            ! Raise pen
            MoveL Offs(next_target, x_offset, y_offset, penup_offset),approach_speed,fine,Alex_Pen_ABB\WObj:=WorkSurface;
        ELSEIF character = "j" THEN
            ! Raise pen to avoid drawing of surface
            position := Lower_J_PtA{1} * font_size;
            next_target.trans := position;
            MoveJ Offs(next_target, x_offset, y_offset, penup_offset),approach_speed,fine,Alex_Pen_ABB\WObj:=WorkSurface;

            ! Drop pen
            MoveL Offs(next_target, x_offset, y_offset, z_offset),approach_speed,fine,Alex_Pen_ABB\WObj:=WorkSurface;

            FOR index FROM 1 TO Dim(Lower_J_PtA, 1) DO
                position := Lower_J_PtA{index} * font_size;
                next_target.trans := position; last_index := index;

                MoveJ Offs(next_target, x_offset, y_offset, z_offset),write_speed,fine,Alex_Pen_ABB\WObj:=WorkSurface;
            ENDFOR

            ! Raise pen
            MoveL Offs(next_target, x_offset, y_offset, penup_offset),approach_speed,fine,Alex_Pen_ABB\WObj:=WorkSurface;

            ! Raise pen to avoid drawing of surface
            position := Lower_J_PtB{1} * font_size;
            next_target.trans := position;
            MoveJ Offs(next_target, x_offset, y_offset, penup_offset),approach_speed,fine,Alex_Pen_ABB\WObj:=WorkSurface;

            ! Drop pen
            MoveL Offs(next_target, x_offset, y_offset, z_offset),approach_speed,fine,Alex_Pen_ABB\WObj:=WorkSurface;

            FOR index FROM 1 TO Dim(Lower_J_PtB, 1) DO
                position := Lower_J_PtB{index} * font_size;
                next_target.trans := position; last_index := index;

                MoveJ Offs(next_target, x_offset, y_offset, z_offset),write_speed,fine,Alex_Pen_ABB\WObj:=WorkSurface;
            ENDFOR

            ! Raise pen
            MoveL Offs(next_target, x_offset, y_offset, penup_offset),approach_speed,fine,Alex_Pen_ABB\WObj:=WorkSurface;
        ELSEIF character = "k" THEN
            ! Raise pen to avoid drawing of surface
            position := Lower_K_PtA{1} * font_size;
            next_target.trans := position;
            MoveJ Offs(next_target, x_offset, y_offset, penup_offset),approach_speed,fine,Alex_Pen_ABB\WObj:=WorkSurface;

            ! Drop pen
            MoveL Offs(next_target, x_offset, y_offset, z_offset),approach_speed,fine,Alex_Pen_ABB\WObj:=WorkSurface;

            FOR index FROM 1 TO Dim(Lower_K_PtA, 1) DO
                position := Lower_K_PtA{index} * font_size;
                next_target.trans := position; last_index := index;

                MoveJ Offs(next_target, x_offset, y_offset, z_offset),write_speed,fine,Alex_Pen_ABB\WObj:=WorkSurface;
            ENDFOR

            ! Raise pen
            MoveL Offs(next_target, x_offset, y_offset, penup_offset),approach_speed,fine,Alex_Pen_ABB\WObj:=WorkSurface;
        ELSEIF character = "l" THEN
            ! Raise pen to avoid drawing of surface
            position := Lower_L_PtA{1} * font_size;
            next_target.trans := position;
            MoveJ Offs(next_target, x_offset, y_offset, penup_offset),approach_speed,fine,Alex_Pen_ABB\WObj:=WorkSurface;

            ! Drop pen
            MoveL Offs(next_target, x_offset, y_offset, z_offset),approach_speed,fine,Alex_Pen_ABB\WObj:=WorkSurface;

            FOR index FROM 1 TO Dim(Lower_L_PtA, 1) DO
                position := Lower_L_PtA{index} * font_size;
                next_target.trans := position; last_index := index;

                MoveJ Offs(next_target, x_offset, y_offset, z_offset),write_speed,fine,Alex_Pen_ABB\WObj:=WorkSurface;
            ENDFOR

            ! Raise pen
            MoveL Offs(next_target, x_offset, y_offset, penup_offset),approach_speed,fine,Alex_Pen_ABB\WObj:=WorkSurface;
        ELSEIF character = "m" THEN
            ! Raise pen to avoid drawing of surface
            position := Lower_M_PtA{1} * font_size;
            next_target.trans := position;
            MoveJ Offs(next_target, x_offset, y_offset, penup_offset),approach_speed,fine,Alex_Pen_ABB\WObj:=WorkSurface;

            ! Drop pen
            MoveL Offs(next_target, x_offset, y_offset, z_offset),approach_speed,fine,Alex_Pen_ABB\WObj:=WorkSurface;

            FOR index FROM 1 TO Dim(Lower_M_PtA, 1) DO
                position := Lower_M_PtA{index} * font_size;
                next_target.trans := position; last_index := index;

                MoveJ Offs(next_target, x_offset, y_offset, z_offset),write_speed,fine,Alex_Pen_ABB\WObj:=WorkSurface;
            ENDFOR

            ! Raise pen
            MoveL Offs(next_target, x_offset, y_offset, penup_offset),approach_speed,fine,Alex_Pen_ABB\WObj:=WorkSurface;
        ELSEIF character = "n" THEN
            ! Raise pen to avoid drawing of surface
            position := Lower_N_PtA{1} * font_size;
            next_target.trans := position;
            MoveJ Offs(next_target, x_offset, y_offset, penup_offset),approach_speed,fine,Alex_Pen_ABB\WObj:=WorkSurface;

            ! Drop pen
            MoveL Offs(next_target, x_offset, y_offset, z_offset),approach_speed,fine,Alex_Pen_ABB\WObj:=WorkSurface;

            FOR index FROM 1 TO Dim(Lower_N_PtA, 1) DO
                position := Lower_N_PtA{index} * font_size;
                next_target.trans := position; last_index := index;

                MoveJ Offs(next_target, x_offset, y_offset, z_offset),write_speed,fine,Alex_Pen_ABB\WObj:=WorkSurface;
            ENDFOR

            ! Raise pen
            MoveL Offs(next_target, x_offset, y_offset, penup_offset),approach_speed,fine,Alex_Pen_ABB\WObj:=WorkSurface;
        ELSEIF character = "o" THEN
            ! Raise pen to avoid drawing of surface
            position := Lower_O_PtA{1} * font_size;
            next_target.trans := position;
            MoveJ Offs(next_target, x_offset, y_offset, penup_offset),approach_speed,fine,Alex_Pen_ABB\WObj:=WorkSurface;

            ! Drop pen
            MoveL Offs(next_target, x_offset, y_offset, z_offset),approach_speed,fine,Alex_Pen_ABB\WObj:=WorkSurface;

            FOR index FROM 1 TO Dim(Lower_O_PtA, 1) DO
                position := Lower_O_PtA{index} * font_size;
                next_target.trans := position; last_index := index;

                MoveJ Offs(next_target, x_offset, y_offset, z_offset),write_speed,fine,Alex_Pen_ABB\WObj:=WorkSurface;
            ENDFOR

            ! Raise pen
            MoveL Offs(next_target, x_offset, y_offset, penup_offset),approach_speed,fine,Alex_Pen_ABB\WObj:=WorkSurface;

            ! Raise pen to avoid drawing of surface
            position := Lower_O_PtB{1} * font_size;
            next_target.trans := position;
            MoveJ Offs(next_target, x_offset, y_offset, penup_offset),approach_speed,fine,Alex_Pen_ABB\WObj:=WorkSurface;

            ! Drop pen
            MoveL Offs(next_target, x_offset, y_offset, z_offset),approach_speed,fine,Alex_Pen_ABB\WObj:=WorkSurface;

            FOR index FROM 1 TO Dim(Lower_O_PtB, 1) DO
                position := Lower_O_PtB{index} * font_size;
                next_target.trans := position; last_index := index;

                MoveJ Offs(next_target, x_offset, y_offset, z_offset),write_speed,fine,Alex_Pen_ABB\WObj:=WorkSurface;
            ENDFOR

            ! Raise pen
            MoveL Offs(next_target, x_offset, y_offset, penup_offset),approach_speed,fine,Alex_Pen_ABB\WObj:=WorkSurface;
        ELSEIF character = "p" THEN
            ! Raise pen to avoid drawing of surface
            position := Lower_P_PtA{1} * font_size;
            next_target.trans := position;
            MoveJ Offs(next_target, x_offset, y_offset, penup_offset),approach_speed,fine,Alex_Pen_ABB\WObj:=WorkSurface;

            ! Drop pen
            MoveL Offs(next_target, x_offset, y_offset, z_offset),approach_speed,fine,Alex_Pen_ABB\WObj:=WorkSurface;

            FOR index FROM 1 TO Dim(Lower_P_PtA, 1) DO
                position := Lower_P_PtA{index} * font_size;
                next_target.trans := position; last_index := index;

                MoveJ Offs(next_target, x_offset, y_offset, z_offset),write_speed,fine,Alex_Pen_ABB\WObj:=WorkSurface;
            ENDFOR

            ! Raise pen
            MoveL Offs(next_target, x_offset, y_offset, penup_offset),approach_speed,fine,Alex_Pen_ABB\WObj:=WorkSurface;

            ! Raise pen to avoid drawing of surface
            position := Lower_P_PtB{1} * font_size;
            next_target.trans := position;
            MoveJ Offs(next_target, x_offset, y_offset, penup_offset),approach_speed,fine,Alex_Pen_ABB\WObj:=WorkSurface;

            ! Drop pen
            MoveL Offs(next_target, x_offset, y_offset, z_offset),approach_speed,fine,Alex_Pen_ABB\WObj:=WorkSurface;

            FOR index FROM 1 TO Dim(Lower_P_PtB, 1) DO
                position := Lower_P_PtB{index} * font_size;
                next_target.trans := position; last_index := index;

                MoveJ Offs(next_target, x_offset, y_offset, z_offset),write_speed,fine,Alex_Pen_ABB\WObj:=WorkSurface;
            ENDFOR

            ! Raise pen
            MoveL Offs(next_target, x_offset, y_offset, penup_offset),approach_speed,fine,Alex_Pen_ABB\WObj:=WorkSurface;
        ELSEIF character = "q" THEN
            ! Raise pen to avoid drawing of surface
            position := Lower_Q_PtA{1} * font_size;
            next_target.trans := position;
            MoveJ Offs(next_target, x_offset, y_offset, penup_offset),approach_speed,fine,Alex_Pen_ABB\WObj:=WorkSurface;

            ! Drop pen
            MoveL Offs(next_target, x_offset, y_offset, z_offset),approach_speed,fine,Alex_Pen_ABB\WObj:=WorkSurface;

            FOR index FROM 1 TO Dim(Lower_Q_PtA, 1) DO
                position := Lower_Q_PtA{index} * font_size;
                next_target.trans := position; last_index := index;

                MoveJ Offs(next_target, x_offset, y_offset, z_offset),write_speed,fine,Alex_Pen_ABB\WObj:=WorkSurface;
            ENDFOR

            ! Raise pen
            MoveL Offs(next_target, x_offset, y_offset, penup_offset),approach_speed,fine,Alex_Pen_ABB\WObj:=WorkSurface;

            ! Raise pen to avoid drawing of surface
            position := Lower_Q_PtB{1} * font_size;
            next_target.trans := position;
            MoveJ Offs(next_target, x_offset, y_offset, penup_offset),approach_speed,fine,Alex_Pen_ABB\WObj:=WorkSurface;

            ! Drop pen
            MoveL Offs(next_target, x_offset, y_offset, z_offset),approach_speed,fine,Alex_Pen_ABB\WObj:=WorkSurface;

            FOR index FROM 1 TO Dim(Lower_Q_PtB, 1) DO
                position := Lower_Q_PtB{index} * font_size;
                next_target.trans := position; last_index := index;

                MoveJ Offs(next_target, x_offset, y_offset, z_offset),write_speed,fine,Alex_Pen_ABB\WObj:=WorkSurface;
            ENDFOR

            ! Raise pen
            MoveL Offs(next_target, x_offset, y_offset, penup_offset),approach_speed,fine,Alex_Pen_ABB\WObj:=WorkSurface;
        ELSEIF character = "r" THEN
            ! Raise pen to avoid drawing of surface
            position := Lower_R_PtA{1} * font_size;
            next_target.trans := position;
            MoveJ Offs(next_target, x_offset, y_offset, penup_offset),approach_speed,fine,Alex_Pen_ABB\WObj:=WorkSurface;

            ! Drop pen
            MoveL Offs(next_target, x_offset, y_offset, z_offset),approach_speed,fine,Alex_Pen_ABB\WObj:=WorkSurface;

            FOR index FROM 1 TO Dim(Lower_R_PtA, 1) DO
                position := Lower_R_PtA{index} * font_size;
                next_target.trans := position; last_index := index;

                MoveJ Offs(next_target, x_offset, y_offset, z_offset),write_speed,fine,Alex_Pen_ABB\WObj:=WorkSurface;
            ENDFOR

            ! Raise pen
            MoveL Offs(next_target, x_offset, y_offset, penup_offset),approach_speed,fine,Alex_Pen_ABB\WObj:=WorkSurface;
        ELSEIF character = "s" THEN
            ! Raise pen to avoid drawing of surface
            position := Lower_S_PtA{1} * font_size;
            next_target.trans := position;
            MoveJ Offs(next_target, x_offset, y_offset, penup_offset),approach_speed,fine,Alex_Pen_ABB\WObj:=WorkSurface;

            ! Drop pen
            MoveL Offs(next_target, x_offset, y_offset, z_offset),approach_speed,fine,Alex_Pen_ABB\WObj:=WorkSurface;

            FOR index FROM 1 TO Dim(Lower_S_PtA, 1) DO
                position := Lower_S_PtA{index} * font_size;
                next_target.trans := position; last_index := index;

                MoveJ Offs(next_target, x_offset, y_offset, z_offset),write_speed,fine,Alex_Pen_ABB\WObj:=WorkSurface;
            ENDFOR

            ! Raise pen
            MoveL Offs(next_target, x_offset, y_offset, penup_offset),approach_speed,fine,Alex_Pen_ABB\WObj:=WorkSurface;
        ELSEIF character = "t" THEN
            ! Raise pen to avoid drawing of surface
            position := Lower_T_PtA{1} * font_size;
            next_target.trans := position;
            MoveJ Offs(next_target, x_offset, y_offset, penup_offset),approach_speed,fine,Alex_Pen_ABB\WObj:=WorkSurface;

            ! Drop pen
            MoveL Offs(next_target, x_offset, y_offset, z_offset),approach_speed,fine,Alex_Pen_ABB\WObj:=WorkSurface;

            FOR index FROM 1 TO Dim(Lower_T_PtA, 1) DO
                position := Lower_T_PtA{index} * font_size;
                next_target.trans := position; last_index := index;

                MoveJ Offs(next_target, x_offset, y_offset, z_offset),write_speed,fine,Alex_Pen_ABB\WObj:=WorkSurface;
            ENDFOR

            ! Raise pen
            MoveL Offs(next_target, x_offset, y_offset, penup_offset),approach_speed,fine,Alex_Pen_ABB\WObj:=WorkSurface;
        ELSEIF character = "u" THEN
            ! Raise pen to avoid drawing of surface
            position := Lower_U_PtA{1} * font_size;
            next_target.trans := position;
            MoveJ Offs(next_target, x_offset, y_offset, penup_offset),approach_speed,fine,Alex_Pen_ABB\WObj:=WorkSurface;

            ! Drop pen
            MoveL Offs(next_target, x_offset, y_offset, z_offset),approach_speed,fine,Alex_Pen_ABB\WObj:=WorkSurface;

            FOR index FROM 1 TO Dim(Lower_U_PtA, 1) DO
                position := Lower_U_PtA{index} * font_size;
                next_target.trans := position; last_index := index;

                MoveJ Offs(next_target, x_offset, y_offset, z_offset),write_speed,fine,Alex_Pen_ABB\WObj:=WorkSurface;
            ENDFOR

            ! Raise pen
            MoveL Offs(next_target, x_offset, y_offset, penup_offset),approach_speed,fine,Alex_Pen_ABB\WObj:=WorkSurface;
        ELSEIF character = "v" THEN
            ! Raise pen to avoid drawing of surface
            position := Lower_V_PtA{1} * font_size;
            next_target.trans := position;
            MoveJ Offs(next_target, x_offset, y_offset, penup_offset),approach_speed,fine,Alex_Pen_ABB\WObj:=WorkSurface;

            ! Drop pen
            MoveL Offs(next_target, x_offset, y_offset, z_offset),approach_speed,fine,Alex_Pen_ABB\WObj:=WorkSurface;

            FOR index FROM 1 TO Dim(Lower_V_PtA, 1) DO
                position := Lower_V_PtA{index} * font_size;
                next_target.trans := position; last_index := index;

                MoveJ Offs(next_target, x_offset, y_offset, z_offset),write_speed,fine,Alex_Pen_ABB\WObj:=WorkSurface;
            ENDFOR

            ! Raise pen
            MoveL Offs(next_target, x_offset, y_offset, penup_offset),approach_speed,fine,Alex_Pen_ABB\WObj:=WorkSurface;
        ELSEIF character = "w" THEN
            ! Raise pen to avoid drawing of surface
            position := Lower_W_PtA{1} * font_size;
            next_target.trans := position;
            MoveJ Offs(next_target, x_offset, y_offset, penup_offset),approach_speed,fine,Alex_Pen_ABB\WObj:=WorkSurface;

            ! Drop pen
            MoveL Offs(next_target, x_offset, y_offset, z_offset),approach_speed,fine,Alex_Pen_ABB\WObj:=WorkSurface;

            FOR index FROM 1 TO Dim(Lower_W_PtA, 1) DO
                position := Lower_W_PtA{index} * font_size;
                next_target.trans := position; last_index := index;

                MoveJ Offs(next_target, x_offset, y_offset, z_offset),write_speed,fine,Alex_Pen_ABB\WObj:=WorkSurface;
            ENDFOR

            ! Raise pen
            MoveL Offs(next_target, x_offset, y_offset, penup_offset),approach_speed,fine,Alex_Pen_ABB\WObj:=WorkSurface;
        ELSEIF character = "x" THEN
            ! Raise pen to avoid drawing of surface
            position := Lower_X_PtA{1} * font_size;
            next_target.trans := position;
            MoveJ Offs(next_target, x_offset, y_offset, penup_offset),approach_speed,fine,Alex_Pen_ABB\WObj:=WorkSurface;

            ! Drop pen
            MoveL Offs(next_target, x_offset, y_offset, z_offset),approach_speed,fine,Alex_Pen_ABB\WObj:=WorkSurface;

            FOR index FROM 1 TO Dim(Lower_X_PtA, 1) DO
                position := Lower_X_PtA{index} * font_size;
                next_target.trans := position; last_index := index;

                MoveJ Offs(next_target, x_offset, y_offset, z_offset),write_speed,fine,Alex_Pen_ABB\WObj:=WorkSurface;
            ENDFOR

            ! Raise pen
            MoveL Offs(next_target, x_offset, y_offset, penup_offset),approach_speed,fine,Alex_Pen_ABB\WObj:=WorkSurface;
        ELSEIF character = "y" THEN
            ! Raise pen to avoid drawing of surface
            position := Lower_Y_PtA{1} * font_size;
            next_target.trans := position;
            MoveJ Offs(next_target, x_offset, y_offset, penup_offset),approach_speed,fine,Alex_Pen_ABB\WObj:=WorkSurface;

            ! Drop pen
            MoveL Offs(next_target, x_offset, y_offset, z_offset),approach_speed,fine,Alex_Pen_ABB\WObj:=WorkSurface;

            FOR index FROM 1 TO Dim(Lower_Y_PtA, 1) DO
                position := Lower_Y_PtA{index} * font_size;
                next_target.trans := position; last_index := index;

                MoveJ Offs(next_target, x_offset, y_offset, z_offset),write_speed,fine,Alex_Pen_ABB\WObj:=WorkSurface;
            ENDFOR

            ! Raise pen
            MoveL Offs(next_target, x_offset, y_offset, penup_offset),approach_speed,fine,Alex_Pen_ABB\WObj:=WorkSurface;
        ELSEIF character = "z" THEN
            ! Raise pen to avoid drawing of surface
            position := Lower_Z_PtA{1} * font_size;
            next_target.trans := position;
            MoveJ Offs(next_target, x_offset, y_offset, penup_offset),approach_speed,fine,Alex_Pen_ABB\WObj:=WorkSurface;

            ! Drop pen
            MoveL Offs(next_target, x_offset, y_offset, z_offset),approach_speed,fine,Alex_Pen_ABB\WObj:=WorkSurface;

            FOR index FROM 1 TO Dim(Lower_Z_PtA, 1) DO
                position := Lower_Z_PtA{index} * font_size;
                next_target.trans := position; last_index := index;

                MoveJ Offs(next_target, x_offset, y_offset, z_offset),write_speed,fine,Alex_Pen_ABB\WObj:=WorkSurface;
            ENDFOR

            ! Raise pen
            MoveL Offs(next_target, x_offset, y_offset, penup_offset),approach_speed,fine,Alex_Pen_ABB\WObj:=WorkSurface;
        ELSEIF character = "{" THEN
            ! Raise pen to avoid drawing of surface
            position := OpenCurlyBrackets_PtA{1} * font_size;
            next_target.trans := position;
            MoveJ Offs(next_target, x_offset, y_offset, penup_offset),approach_speed,fine,Alex_Pen_ABB\WObj:=WorkSurface;

            ! Drop pen
            MoveL Offs(next_target, x_offset, y_offset, z_offset),approach_speed,fine,Alex_Pen_ABB\WObj:=WorkSurface;

            FOR index FROM 1 TO Dim(OpenCurlyBrackets_PtA, 1) DO
                position := OpenCurlyBrackets_PtA{index} * font_size;
                next_target.trans := position; last_index := index;

                MoveJ Offs(next_target, x_offset, y_offset, z_offset),write_speed,fine,Alex_Pen_ABB\WObj:=WorkSurface;
            ENDFOR

            ! Raise pen
            MoveL Offs(next_target, x_offset, y_offset, penup_offset),approach_speed,fine,Alex_Pen_ABB\WObj:=WorkSurface;
        ELSEIF character = "}" THEN
            ! Raise pen to avoid drawing of surface
            position := CloseCurlyBrackets_PtB{1} * font_size;
            next_target.trans := position;
            MoveJ Offs(next_target, x_offset, y_offset, penup_offset),approach_speed,fine,Alex_Pen_ABB\WObj:=WorkSurface;

            ! Drop pen
            MoveL Offs(next_target, x_offset, y_offset, z_offset),approach_speed,fine,Alex_Pen_ABB\WObj:=WorkSurface;

            FOR index FROM 1 TO Dim(CloseCurlyBrackets_PtB, 1) DO
                position := CloseCurlyBrackets_PtB{index} * font_size;
                next_target.trans := position; last_index := index;

                MoveJ Offs(next_target, x_offset, y_offset, z_offset),write_speed,fine,Alex_Pen_ABB\WObj:=WorkSurface;
            ENDFOR

            ! Raise pen
            MoveL Offs(next_target, x_offset, y_offset, penup_offset),approach_speed,fine,Alex_Pen_ABB\WObj:=WorkSurface;
        ELSEIF character = "|" THEN
            ! Raise pen to avoid drawing of surface
            position := VerticalBar_PtA{1} * font_size;
            next_target.trans := position;
            MoveJ Offs(next_target, x_offset, y_offset, penup_offset),approach_speed,fine,Alex_Pen_ABB\WObj:=WorkSurface;

            ! Drop pen
            MoveL Offs(next_target, x_offset, y_offset, z_offset),approach_speed,fine,Alex_Pen_ABB\WObj:=WorkSurface;

            FOR index FROM 1 TO Dim(VerticalBar_PtA, 1) DO
                position := VerticalBar_PtA{index} * font_size;
                next_target.trans := position; last_index := index;

                MoveJ Offs(next_target, x_offset, y_offset, z_offset),write_speed,fine,Alex_Pen_ABB\WObj:=WorkSurface;
            ENDFOR

            ! Raise pen
            MoveL Offs(next_target, x_offset, y_offset, penup_offset),approach_speed,fine,Alex_Pen_ABB\WObj:=WorkSurface;
        ELSEIF character = "~" THEN
            ! Raise pen to avoid drawing of surface
            position := Tilty_PtA{1} * font_size;
            next_target.trans := position;
            MoveJ Offs(next_target, x_offset, y_offset, penup_offset),approach_speed,fine,Alex_Pen_ABB\WObj:=WorkSurface;

            ! Drop pen
            MoveL Offs(next_target, x_offset, y_offset, z_offset),approach_speed,fine,Alex_Pen_ABB\WObj:=WorkSurface;

            FOR index FROM 1 TO Dim(Tilty_PtA, 1) DO
                position := Tilty_PtA{index} * font_size;
                next_target.trans := position; last_index := index;

                MoveJ Offs(next_target, x_offset, y_offset, z_offset),write_speed,fine,Alex_Pen_ABB\WObj:=WorkSurface;
            ENDFOR

            ! Raise pen
            MoveL Offs(next_target, x_offset, y_offset, penup_offset),approach_speed,fine,Alex_Pen_ABB\WObj:=WorkSurface;
        ELSE
            TPWrite "Unknown character " + character;
        ENDIF

    ENDPROC


    !***********************************************************
    !
    ! Procedure DrawArtWork_House
    !   This procedure draws my house artwork on the work surface
    !   This is mainly used by the Special User function
    !
    ! Example
    !   VAR speeddata approach_speed := v100;  // Approach speed for arm
    !   VAR speeddata write_speed := v80;      // Write speed for arm
    !   VAR num x_offset := 0;                 // x offset from worksurface origin
    !   VAR num y_offset := 0;                 // y offset from worksurface origin
    !   VAR num z_offset := 0;                 // z offset from worksurface origin
    !   VAR num pen_offset := 30;              // Defines pen position for pen up
    !
    !   DrawArtWork_House 1.0, approach_speed, write_speed, x_offset, y_offset, z_offset, penup_offset;
    !
    !***********************************************************
    PROC DrawArtWork_House(num font_size, speeddata approach_speed, speeddata write_speed, num x_offset, num y_offset, num z_offset, num penup_offset)
        ! Define all points for artwork
        VAR pos pos0{30} := [[147.0, 28.0, 0],[146.0, 29.0, 0],[146.0, 48.0, 0],[147.0, 49.0, 0],[147.0, 60.0, 0],[148.0, 61.0, 0],[148.0, 67.0, 0],[149.0, 68.0, 0],[149.0, 77.0, 0],[151.0, 79.0, 0],[153.0, 79.0, 0],[154.0, 78.0, 0],[155.0, 78.0, 0],[156.0, 77.0, 0],[156.0, 72.0, 0],[155.0, 71.0, 0],[155.0, 67.0, 0],[154.0, 66.0, 0],[154.0, 60.0, 0],[153.0, 59.0, 0],[153.0, 16.0, 0],[154.0, 15.0, 0],[154.0, 13.0, 0],[151.0, 10.0, 0],[150.0, 10.0, 0],[148.0, 12.0, 0],[148.0, 14.0, 0],[147.0, 15.0, 0],[147.0, 28.0, 0],[146.0, 29.0, 0]];
        VAR pos pos1{120} := [[99.0, 127.0, 0],[98.0, 128.0, 0],[98.0, 129.0, 0],[101.0, 132.0, 0],[102.0, 131.0, 0],[103.0, 131.0, 0],[106.0, 128.0, 0],[107.0, 128.0, 0],[110.0, 125.0, 0],[111.0, 125.0, 0],[114.0, 122.0, 0],[115.0, 122.0, 0],[118.0, 119.0, 0],[119.0, 119.0, 0],[121.0, 117.0, 0],[122.0, 117.0, 0],[125.0, 114.0, 0],[126.0, 114.0, 0],[129.0, 111.0, 0],[130.0, 111.0, 0],[131.0, 110.0, 0],[132.0, 110.0, 0],[134.0, 108.0, 0],[135.0, 108.0, 0],[138.0, 105.0, 0],[139.0, 105.0, 0],[140.0, 104.0, 0],[141.0, 104.0, 0],[142.0, 103.0, 0],[143.0, 103.0, 0],[146.0, 100.0, 0],[147.0, 100.0, 0],[148.0, 99.0, 0],[149.0, 99.0, 0],[151.0, 97.0, 0],[152.0, 97.0, 0],[153.0, 96.0, 0],[154.0, 96.0, 0],[156.0, 94.0, 0],[158.0, 94.0, 0],[159.0, 93.0, 0],[159.0, 92.0, 0],[161.0, 92.0, 0],[164.0, 89.0, 0],[166.0, 89.0, 0],[168.0, 87.0, 0],[169.0, 87.0, 0],[170.0, 86.0, 0],[172.0, 86.0, 0],[175.0, 83.0, 0],[177.0, 83.0, 0],[179.0, 81.0, 0],[180.0, 81.0, 0],[181.0, 80.0, 0],[183.0, 80.0, 0],[184.0, 79.0, 0],[184.0, 78.0, 0],[186.0, 78.0, 0],[187.0, 77.0, 0],[187.0, 76.0, 0],[184.0, 73.0, 0],[182.0, 73.0, 0],[181.0, 74.0, 0],[179.0, 74.0, 0],[177.0, 76.0, 0],[176.0, 76.0, 0],[175.0, 77.0, 0],[173.0, 77.0, 0],[172.0, 78.0, 0],[172.0, 79.0, 0],[170.0, 79.0, 0],[169.0, 80.0, 0],[168.0, 80.0, 0],[166.0, 82.0, 0],[164.0, 82.0, 0],[162.0, 84.0, 0],[161.0, 84.0, 0],[160.0, 85.0, 0],[159.0, 85.0, 0],[156.0, 88.0, 0],[154.0, 88.0, 0],[151.0, 91.0, 0],[150.0, 91.0, 0],[149.0, 92.0, 0],[148.0, 92.0, 0],[147.0, 93.0, 0],[146.0, 93.0, 0],[143.0, 96.0, 0],[141.0, 96.0, 0],[138.0, 99.0, 0],[136.0, 99.0, 0],[135.0, 100.0, 0],[135.0, 101.0, 0],[134.0, 101.0, 0],[133.0, 102.0, 0],[132.0, 102.0, 0],[130.0, 104.0, 0],[129.0, 104.0, 0],[126.0, 107.0, 0],[125.0, 107.0, 0],[124.0, 108.0, 0],[123.0, 108.0, 0],[121.0, 110.0, 0],[120.0, 110.0, 0],[119.0, 111.0, 0],[119.0, 112.0, 0],[118.0, 112.0, 0],[117.0, 113.0, 0],[116.0, 113.0, 0],[113.0, 116.0, 0],[112.0, 116.0, 0],[110.0, 118.0, 0],[109.0, 118.0, 0],[105.0, 122.0, 0],[104.0, 122.0, 0],[102.0, 124.0, 0],[101.0, 124.0, 0],[99.0, 126.0, 0],[99.0, 127.0, 0],[98.0, 128.0, 0]];
        VAR pos pos2{51} := [[78.0, 87.0, 0],[78.0, 89.0, 0],[79.0, 90.0, 0],[80.0, 90.0, 0],[81.0, 91.0, 0],[82.0, 91.0, 0],[83.0, 92.0, 0],[83.0, 93.0, 0],[84.0, 94.0, 0],[84.0, 95.0, 0],[85.0, 96.0, 0],[85.0, 97.0, 0],[90.0, 102.0, 0],[91.0, 102.0, 0],[92.0, 103.0, 0],[93.0, 103.0, 0],[94.0, 104.0, 0],[96.0, 104.0, 0],[97.0, 105.0, 0],[103.0, 105.0, 0],[104.0, 104.0, 0],[105.0, 104.0, 0],[106.0, 103.0, 0],[109.0, 103.0, 0],[112.0, 100.0, 0],[113.0, 100.0, 0],[114.0, 99.0, 0],[114.0, 97.0, 0],[115.0, 97.0, 0],[116.0, 96.0, 0],[116.0, 95.0, 0],[117.0, 94.0, 0],[117.0, 92.0, 0],[118.0, 92.0, 0],[119.0, 91.0, 0],[121.0, 91.0, 0],[122.0, 90.0, 0],[122.0, 87.0, 0],[121.0, 86.0, 0],[118.0, 86.0, 0],[117.0, 87.0, 0],[111.0, 87.0, 0],[110.0, 88.0, 0],[95.0, 88.0, 0],[94.0, 87.0, 0],[86.0, 87.0, 0],[85.0, 86.0, 0],[81.0, 86.0, 0],[80.0, 85.0, 0],[78.0, 87.0, 0],[78.0, 89.0, 0]];
        VAR pos pos3{12} := [[88.0, 92.0, 0],[112.0, 92.0, 0],[112.0, 93.0, 0],[110.0, 95.0, 0],[110.0, 96.0, 0],[109.0, 96.0, 0],[106.0, 99.0, 0],[94.0, 99.0, 0],[89.0, 94.0, 0],[89.0, 93.0, 0],[88.0, 92.0, 0],[112.0, 92.0, 0]];
        VAR pos pos4{46} := [[78.0, 70.0, 0],[77.0, 71.0, 0],[78.0, 72.0, 0],[79.0, 72.0, 0],[80.0, 73.0, 0],[81.0, 72.0, 0],[81.0, 70.0, 0],[82.0, 69.0, 0],[90.0, 69.0, 0],[91.0, 68.0, 0],[113.0, 68.0, 0],[114.0, 69.0, 0],[127.0, 69.0, 0],[127.0, 71.0, 0],[128.0, 72.0, 0],[129.0, 72.0, 0],[130.0, 73.0, 0],[131.0, 72.0, 0],[131.0, 60.0, 0],[130.0, 59.0, 0],[130.0, 47.0, 0],[129.0, 46.0, 0],[129.0, 36.0, 0],[130.0, 35.0, 0],[130.0, 25.0, 0],[129.0, 24.0, 0],[128.0, 24.0, 0],[126.0, 26.0, 0],[126.0, 27.0, 0],[125.0, 28.0, 0],[122.0, 28.0, 0],[121.0, 29.0, 0],[88.0, 29.0, 0],[87.0, 28.0, 0],[85.0, 28.0, 0],[84.0, 27.0, 0],[84.0, 26.0, 0],[82.0, 24.0, 0],[81.0, 24.0, 0],[80.0, 25.0, 0],[80.0, 59.0, 0],[79.0, 60.0, 0],[79.0, 65.0, 0],[78.0, 66.0, 0],[78.0, 70.0, 0],[77.0, 71.0, 0]];
        VAR pos pos5{31} := [[106.0, 35.0, 0],[107.0, 34.0, 0],[107.0, 33.0, 0],[116.0, 33.0, 0],[117.0, 32.0, 0],[125.0, 32.0, 0],[126.0, 33.0, 0],[126.0, 38.0, 0],[125.0, 39.0, 0],[125.0, 45.0, 0],[126.0, 46.0, 0],[126.0, 57.0, 0],[127.0, 58.0, 0],[127.0, 65.0, 0],[110.0, 65.0, 0],[109.0, 64.0, 0],[108.0, 64.0, 0],[107.0, 63.0, 0],[107.0, 60.0, 0],[106.0, 59.0, 0],[106.0, 52.0, 0],[108.0, 50.0, 0],[124.0, 50.0, 0],[125.0, 49.0, 0],[125.0, 48.0, 0],[124.0, 47.0, 0],[119.0, 47.0, 0],[118.0, 46.0, 0],[106.0, 46.0, 0],[106.0, 35.0, 0],[107.0, 34.0, 0]];
        VAR pos pos6{30} := [[83.0, 52.0, 0],[84.0, 51.0, 0],[84.0, 33.0, 0],[85.0, 32.0, 0],[92.0, 32.0, 0],[93.0, 33.0, 0],[102.0, 33.0, 0],[103.0, 34.0, 0],[103.0, 39.0, 0],[102.0, 40.0, 0],[102.0, 43.0, 0],[103.0, 44.0, 0],[103.0, 45.0, 0],[102.0, 46.0, 0],[91.0, 46.0, 0],[90.0, 47.0, 0],[85.0, 47.0, 0],[84.0, 48.0, 0],[84.0, 49.0, 0],[85.0, 50.0, 0],[102.0, 50.0, 0],[102.0, 51.0, 0],[103.0, 52.0, 0],[103.0, 63.0, 0],[102.0, 64.0, 0],[98.0, 64.0, 0],[97.0, 65.0, 0],[83.0, 65.0, 0],[83.0, 52.0, 0],[84.0, 51.0, 0]];
        VAR pos pos7{26} := [[54.0, 69.0, 0],[53.0, 70.0, 0],[53.0, 74.0, 0],[54.0, 75.0, 0],[58.0, 75.0, 0],[59.0, 74.0, 0],[59.0, 71.0, 0],[60.0, 70.0, 0],[60.0, 66.0, 0],[61.0, 65.0, 0],[61.0, 54.0, 0],[62.0, 53.0, 0],[62.0, 45.0, 0],[63.0, 44.0, 0],[63.0, 12.0, 0],[61.0, 10.0, 0],[58.0, 10.0, 0],[57.0, 11.0, 0],[57.0, 45.0, 0],[56.0, 46.0, 0],[56.0, 53.0, 0],[55.0, 54.0, 0],[55.0, 59.0, 0],[54.0, 60.0, 0],[54.0, 69.0, 0],[53.0, 70.0, 0]];
        VAR pos pos8{107} := [[33.0, 68.0, 0],[32.0, 69.0, 0],[32.0, 71.0, 0],[33.0, 72.0, 0],[34.0, 72.0, 0],[37.0, 75.0, 0],[38.0, 75.0, 0],[38.0, 76.0, 0],[42.0, 80.0, 0],[43.0, 80.0, 0],[63.0, 100.0, 0],[63.0, 101.0, 0],[65.0, 103.0, 0],[66.0, 103.0, 0],[66.0, 104.0, 0],[67.0, 105.0, 0],[68.0, 105.0, 0],[68.0, 106.0, 0],[71.0, 109.0, 0],[71.0, 110.0, 0],[72.0, 111.0, 0],[73.0, 111.0, 0],[74.0, 112.0, 0],[74.0, 113.0, 0],[77.0, 116.0, 0],[77.0, 117.0, 0],[79.0, 119.0, 0],[80.0, 119.0, 0],[80.0, 121.0, 0],[81.0, 122.0, 0],[82.0, 122.0, 0],[82.0, 124.0, 0],[83.0, 125.0, 0],[84.0, 125.0, 0],[85.0, 126.0, 0],[85.0, 127.0, 0],[88.0, 130.0, 0],[88.0, 131.0, 0],[89.0, 132.0, 0],[90.0, 132.0, 0],[91.0, 131.0, 0],[92.0, 131.0, 0],[93.0, 130.0, 0],[93.0, 128.0, 0],[92.0, 127.0, 0],[92.0, 125.0, 0],[91.0, 124.0, 0],[90.0, 124.0, 0],[90.0, 123.0, 0],[88.0, 121.0, 0],[88.0, 120.0, 0],[83.0, 115.0, 0],[83.0, 114.0, 0],[81.0, 112.0, 0],[81.0, 111.0, 0],[80.0, 110.0, 0],[79.0, 110.0, 0],[78.0, 109.0, 0],[78.0, 108.0, 0],[74.0, 104.0, 0],[74.0, 103.0, 0],[73.0, 102.0, 0],[72.0, 102.0, 0],[72.0, 101.0, 0],[70.0, 99.0, 0],[69.0, 99.0, 0],[69.0, 98.0, 0],[67.0, 96.0, 0],[67.0, 95.0, 0],[65.0, 93.0, 0],[64.0, 93.0, 0],[64.0, 92.0, 0],[63.0, 91.0, 0],[62.0, 91.0, 0],[61.0, 90.0, 0],[61.0, 89.0, 0],[60.0, 88.0, 0],[59.0, 88.0, 0],[58.0, 87.0, 0],[58.0, 86.0, 0],[57.0, 85.0, 0],[56.0, 85.0, 0],[55.0, 84.0, 0],[55.0, 83.0, 0],[54.0, 82.0, 0],[53.0, 82.0, 0],[53.0, 81.0, 0],[51.0, 79.0, 0],[50.0, 79.0, 0],[50.0, 78.0, 0],[49.0, 77.0, 0],[48.0, 77.0, 0],[47.0, 76.0, 0],[47.0, 75.0, 0],[46.0, 74.0, 0],[44.0, 74.0, 0],[44.0, 73.0, 0],[42.0, 71.0, 0],[41.0, 71.0, 0],[41.0, 70.0, 0],[39.0, 68.0, 0],[38.0, 68.0, 0],[37.0, 67.0, 0],[35.0, 67.0, 0],[34.0, 68.0, 0],[33.0, 68.0, 0],[32.0, 69.0, 0]];
        VAR pos pos9{54} := [[0.0, 2.0, 0],[0.0, 4.0, 0],[2.0, 6.0, 0],[4.0, 6.0, 0],[5.0, 7.0, 0],[10.0, 7.0, 0],[11.0, 8.0, 0],[27.0, 8.0, 0],[28.0, 9.0, 0],[46.0, 9.0, 0],[47.0, 10.0, 0],[71.0, 10.0, 0],[72.0, 9.0, 0],[100.0, 9.0, 0],[101.0, 8.0, 0],[185.0, 8.0, 0],[186.0, 9.0, 0],[193.0, 9.0, 0],[194.0, 10.0, 0],[199.0, 10.0, 0],[200.0, 11.0, 0],[208.0, 11.0, 0],[209.0, 10.0, 0],[209.0, 6.0, 0],[208.0, 5.0, 0],[206.0, 5.0, 0],[205.0, 4.0, 0],[194.0, 4.0, 0],[193.0, 3.0, 0],[185.0, 3.0, 0],[184.0, 2.0, 0],[172.0, 2.0, 0],[171.0, 1.0, 0],[122.0, 1.0, 0],[121.0, 2.0, 0],[117.0, 2.0, 0],[116.0, 1.0, 0],[106.0, 1.0, 0],[105.0, 2.0, 0],[92.0, 2.0, 0],[91.0, 3.0, 0],[70.0, 3.0, 0],[69.0, 4.0, 0],[47.0, 4.0, 0],[46.0, 3.0, 0],[29.0, 3.0, 0],[28.0, 2.0, 0],[19.0, 2.0, 0],[18.0, 1.0, 0],[5.0, 1.0, 0],[4.0, 0.0, 0],[2.0, 0.0, 0],[0.0, 2.0, 0],[0.0, 4.0, 0]];

        ! Define variables to be used while drawing
        VAR pos position := [0,0,0];
        VAR robtarget next_target := [[0,0,0],[0,0,1,0],[0,0,0,0],[9E+09,9E+09,9E+09,9E+09,9E+09,9E+09]];

        ! Update the penup_offset based on the z_offset
        penup_offset := z_offset + penup_offset;

        ! Raise pen to avoid drawing of surface while moving to the new approach position
        position := pos0{1} * font_size;
        next_target.trans := position;
        MoveJ Offs(next_target, x_offset, y_offset, penup_offset),approach_speed,fine,Alex_Pen_ABB\WObj:=WorkSurface;

        ! Drop pen
        MoveL Offs(next_target, x_offset, y_offset, z_offset),approach_speed,fine,Alex_Pen_ABB\WObj:=WorkSurface;

        FOR index FROM 1 TO Dim(pos0, 1) DO
            position := pos0{index} * font_size;
            next_target.trans := position;

            MoveL Offs(next_target, x_offset, y_offset, z_offset),approach_speed,fine,Alex_Pen_ABB\WObj:=WorkSurface;
        ENDFOR

        ! Raise pen
        MoveL Offs(next_target, x_offset, y_offset, penup_offset),approach_speed,fine,Alex_Pen_ABB\WObj:=WorkSurface;

        ! Raise pen to avoid drawing of surface while moving to the new approach position
        position := pos1{1} * font_size;
        next_target.trans := position;
        MoveJ Offs(next_target, x_offset, y_offset, penup_offset),approach_speed,fine,Alex_Pen_ABB\WObj:=WorkSurface;

        ! Drop pen
        MoveL Offs(next_target, x_offset, y_offset, z_offset),approach_speed,fine,Alex_Pen_ABB\WObj:=WorkSurface;

        FOR index FROM 1 TO Dim(pos1, 1) DO
            position := pos1{index} * font_size;
            next_target.trans := position;

            MoveL Offs(next_target, x_offset, y_offset, z_offset),approach_speed,fine,Alex_Pen_ABB\WObj:=WorkSurface;
        ENDFOR

        ! Raise pen
        MoveL Offs(next_target, x_offset, y_offset, penup_offset),approach_speed,fine,Alex_Pen_ABB\WObj:=WorkSurface;

        ! Raise pen to avoid drawing of surface while moving to the new approach position
        position := pos2{1} * font_size;
        next_target.trans := position;
        MoveJ Offs(next_target, x_offset, y_offset, penup_offset),approach_speed,fine,Alex_Pen_ABB\WObj:=WorkSurface;

        ! Drop pen
        MoveL Offs(next_target, x_offset, y_offset, z_offset),approach_speed,fine,Alex_Pen_ABB\WObj:=WorkSurface;

        FOR index FROM 1 TO Dim(pos2, 1) DO
            position := pos2{index} * font_size;
            next_target.trans := position;

            MoveL Offs(next_target, x_offset, y_offset, z_offset),approach_speed,fine,Alex_Pen_ABB\WObj:=WorkSurface;
        ENDFOR

        ! Raise pen
        MoveL Offs(next_target, x_offset, y_offset, penup_offset),approach_speed,fine,Alex_Pen_ABB\WObj:=WorkSurface;

        ! Raise pen to avoid drawing of surface while moving to the new approach position
        position := pos3{1} * font_size;
        next_target.trans := position;
        MoveJ Offs(next_target, x_offset, y_offset, penup_offset),approach_speed,fine,Alex_Pen_ABB\WObj:=WorkSurface;

        ! Drop pen
        MoveL Offs(next_target, x_offset, y_offset, z_offset),approach_speed,fine,Alex_Pen_ABB\WObj:=WorkSurface;

        FOR index FROM 1 TO Dim(pos3, 1) DO
            position := pos3{index} * font_size;
            next_target.trans := position;

            MoveL Offs(next_target, x_offset, y_offset, z_offset),approach_speed,fine,Alex_Pen_ABB\WObj:=WorkSurface;
        ENDFOR

        ! Raise pen
        MoveL Offs(next_target, x_offset, y_offset, penup_offset),approach_speed,fine,Alex_Pen_ABB\WObj:=WorkSurface;

        ! Raise pen to avoid drawing of surface while moving to the new approach position
        position := pos4{1} * font_size;
        next_target.trans := position;
        MoveJ Offs(next_target, x_offset, y_offset, penup_offset),approach_speed,fine,Alex_Pen_ABB\WObj:=WorkSurface;

        ! Drop pen
        MoveL Offs(next_target, x_offset, y_offset, z_offset),approach_speed,fine,Alex_Pen_ABB\WObj:=WorkSurface;

        FOR index FROM 1 TO Dim(pos4, 1) DO
            position := pos4{index} * font_size;
            next_target.trans := position;

            MoveL Offs(next_target, x_offset, y_offset, z_offset),approach_speed,fine,Alex_Pen_ABB\WObj:=WorkSurface;
        ENDFOR

        ! Raise pen
        MoveL Offs(next_target, x_offset, y_offset, penup_offset),approach_speed,fine,Alex_Pen_ABB\WObj:=WorkSurface;

        ! Raise pen to avoid drawing of surface while moving to the new approach position
        position := pos5{1} * font_size;
        next_target.trans := position;
        MoveJ Offs(next_target, x_offset, y_offset, penup_offset),approach_speed,fine,Alex_Pen_ABB\WObj:=WorkSurface;

        ! Drop pen
        MoveL Offs(next_target, x_offset, y_offset, z_offset),approach_speed,fine,Alex_Pen_ABB\WObj:=WorkSurface;

        FOR index FROM 1 TO Dim(pos5, 1) DO
            position := pos5{index} * font_size;
            next_target.trans := position;

            MoveL Offs(next_target, x_offset, y_offset, z_offset),approach_speed,fine,Alex_Pen_ABB\WObj:=WorkSurface;
        ENDFOR

        ! Raise pen
        MoveL Offs(next_target, x_offset, y_offset, penup_offset),approach_speed,fine,Alex_Pen_ABB\WObj:=WorkSurface;

        ! Raise pen to avoid drawing of surface while moving to the new approach position
        position := pos6{1} * font_size;
        next_target.trans := position;
        MoveJ Offs(next_target, x_offset, y_offset, penup_offset),approach_speed,fine,Alex_Pen_ABB\WObj:=WorkSurface;

        ! Drop pen
        MoveL Offs(next_target, x_offset, y_offset, z_offset),approach_speed,fine,Alex_Pen_ABB\WObj:=WorkSurface;

        FOR index FROM 1 TO Dim(pos6, 1) DO
            position := pos6{index} * font_size;
            next_target.trans := position;

            MoveL Offs(next_target, x_offset, y_offset, z_offset),approach_speed,fine,Alex_Pen_ABB\WObj:=WorkSurface;
        ENDFOR

        ! Raise pen
        MoveL Offs(next_target, x_offset, y_offset, penup_offset),approach_speed,fine,Alex_Pen_ABB\WObj:=WorkSurface;

        ! Raise pen to avoid drawing of surface while moving to the new approach position
        position := pos7{1} * font_size;
        next_target.trans := position;
        MoveJ Offs(next_target, x_offset, y_offset, penup_offset),approach_speed,fine,Alex_Pen_ABB\WObj:=WorkSurface;

        ! Drop pen
        MoveL Offs(next_target, x_offset, y_offset, z_offset),approach_speed,fine,Alex_Pen_ABB\WObj:=WorkSurface;

        FOR index FROM 1 TO Dim(pos7, 1) DO
            position := pos7{index} * font_size;
            next_target.trans := position;

            MoveL Offs(next_target, x_offset, y_offset, z_offset),approach_speed,fine,Alex_Pen_ABB\WObj:=WorkSurface;
        ENDFOR

        ! Raise pen
        MoveL Offs(next_target, x_offset, y_offset, penup_offset),approach_speed,fine,Alex_Pen_ABB\WObj:=WorkSurface;

        ! Raise pen to avoid drawing of surface while moving to the new approach position
        position := pos8{1} * font_size;
        next_target.trans := position;
        MoveJ Offs(next_target, x_offset, y_offset, penup_offset),approach_speed,fine,Alex_Pen_ABB\WObj:=WorkSurface;

        ! Drop pen
        MoveL Offs(next_target, x_offset, y_offset, z_offset),approach_speed,fine,Alex_Pen_ABB\WObj:=WorkSurface;

        FOR index FROM 1 TO Dim(pos8, 1) DO
            position := pos8{index} * font_size;
            next_target.trans := position;

            MoveL Offs(next_target, x_offset, y_offset, z_offset),approach_speed,fine,Alex_Pen_ABB\WObj:=WorkSurface;
        ENDFOR

        ! Raise pen
        MoveL Offs(next_target, x_offset, y_offset, penup_offset),approach_speed,fine,Alex_Pen_ABB\WObj:=WorkSurface;

        ! Raise pen to avoid drawing of surface while moving to the new approach position
        position := pos9{1} * font_size;
        next_target.trans := position;
        MoveJ Offs(next_target, x_offset, y_offset, penup_offset),approach_speed,fine,Alex_Pen_ABB\WObj:=WorkSurface;

        ! Drop pen
        MoveL Offs(next_target, x_offset, y_offset, z_offset),approach_speed,fine,Alex_Pen_ABB\WObj:=WorkSurface;

        FOR index FROM 1 TO Dim(pos9, 1) DO
            position := pos9{index} * font_size;
            next_target.trans := position;

            MoveL Offs(next_target, x_offset, y_offset, z_offset),approach_speed,fine,Alex_Pen_ABB\WObj:=WorkSurface;
        ENDFOR

        ! Raise pen
        MoveL Offs(next_target, x_offset, y_offset, penup_offset),approach_speed,fine,Alex_Pen_ABB\WObj:=WorkSurface;

    ENDPROC

    !***********************************************************
    !
    ! Procedure DrawArtWork_Glasses
    !   This procedure draws my glasses artwork on the work surface
    !   This is mainly used by the Special User function
    !
    ! Example
    !   VAR speeddata approach_speed := v100;  // Approach speed for arm
    !   VAR speeddata write_speed := v80;      // Write speed for arm
    !   VAR num x_offset := 0;                 // x offset from worksurface origin
    !   VAR num y_offset := 0;                 // y offset from worksurface origin
    !   VAR num z_offset := 0;                 // z offset from worksurface origin
    !   VAR num pen_offset := 30;              // Defines pen position for pen up
    !
    !   DrawArtWork_Glasses 1.0, approach_speed, write_speed, x_offset, y_offset, z_offset, penup_offset;
    !
    !***********************************************************
    PROC DrawArtWork_Glasses(num font_size, speeddata approach_speed, speeddata write_speed, num x_offset, num y_offset, num z_offset, num penup_offset)
        ! Define all points for artwork
        VAR pos pos0{233} := [[1.0, 42.0, 0],[0.0, 43.0, 0],[0.0, 47.0, 0],[1.0, 48.0, 0],[1.0, 49.0, 0],[5.0, 53.0, 0],[5.0, 54.0, 0],[9.0, 58.0, 0],[9.0, 59.0, 0],[10.0, 60.0, 0],[10.0, 61.0, 0],[11.0, 62.0, 0],[11.0, 63.0, 0],[12.0, 64.0, 0],[12.0, 65.0, 0],[14.0, 67.0, 0],[14.0, 68.0, 0],[22.0, 76.0, 0],[23.0, 76.0, 0],[24.0, 77.0, 0],[25.0, 77.0, 0],[26.0, 78.0, 0],[27.0, 78.0, 0],[28.0, 79.0, 0],[30.0, 79.0, 0],[31.0, 80.0, 0],[35.0, 80.0, 0],[36.0, 81.0, 0],[41.0, 81.0, 0],[42.0, 82.0, 0],[50.0, 82.0, 0],[51.0, 83.0, 0],[63.0, 83.0, 0],[64.0, 84.0, 0],[65.0, 84.0, 0],[66.0, 83.0, 0],[67.0, 83.0, 0],[68.0, 84.0, 0],[128.0, 84.0, 0],[129.0, 83.0, 0],[130.0, 84.0, 0],[132.0, 84.0, 0],[133.0, 83.0, 0],[134.0, 84.0, 0],[135.0, 84.0, 0],[136.0, 83.0, 0],[162.0, 83.0, 0],[163.0, 82.0, 0],[164.0, 82.0, 0],[165.0, 83.0, 0],[166.0, 82.0, 0],[171.0, 82.0, 0],[172.0, 81.0, 0],[176.0, 81.0, 0],[177.0, 80.0, 0],[180.0, 80.0, 0],[181.0, 79.0, 0],[183.0, 79.0, 0],[184.0, 78.0, 0],[185.0, 78.0, 0],[186.0, 77.0, 0],[187.0, 77.0, 0],[188.0, 76.0, 0],[189.0, 76.0, 0],[197.0, 68.0, 0],[197.0, 67.0, 0],[198.0, 66.0, 0],[198.0, 65.0, 0],[199.0, 64.0, 0],[199.0, 63.0, 0],[200.0, 62.0, 0],[200.0, 61.0, 0],[202.0, 59.0, 0],[202.0, 58.0, 0],[205.0, 55.0, 0],[205.0, 54.0, 0],[209.0, 50.0, 0],[209.0, 48.0, 0],[210.0, 47.0, 0],[210.0, 43.0, 0],[209.0, 42.0, 0],[209.0, 40.0, 0],[202.0, 33.0, 0],[202.0, 32.0, 0],[201.0, 31.0, 0],[201.0, 29.0, 0],[200.0, 28.0, 0],[200.0, 26.0, 0],[199.0, 25.0, 0],[199.0, 24.0, 0],[198.0, 23.0, 0],[198.0, 21.0, 0],[196.0, 19.0, 0],[196.0, 18.0, 0],[195.0, 17.0, 0],[195.0, 16.0, 0],[193.0, 14.0, 0],[193.0, 13.0, 0],[186.0, 6.0, 0],[185.0, 6.0, 0],[183.0, 4.0, 0],[182.0, 4.0, 0],[181.0, 3.0, 0],[180.0, 3.0, 0],[179.0, 2.0, 0],[177.0, 2.0, 0],[176.0, 1.0, 0],[173.0, 1.0, 0],[172.0, 0.0, 0],[163.0, 0.0, 0],[162.0, 1.0, 0],[158.0, 1.0, 0],[157.0, 2.0, 0],[155.0, 2.0, 0],[154.0, 3.0, 0],[153.0, 3.0, 0],[152.0, 4.0, 0],[150.0, 4.0, 0],[148.0, 6.0, 0],[147.0, 6.0, 0],[146.0, 7.0, 0],[145.0, 7.0, 0],[144.0, 8.0, 0],[143.0, 8.0, 0],[140.0, 11.0, 0],[139.0, 11.0, 0],[127.0, 23.0, 0],[127.0, 24.0, 0],[125.0, 26.0, 0],[125.0, 27.0, 0],[123.0, 29.0, 0],[123.0, 30.0, 0],[121.0, 32.0, 0],[121.0, 34.0, 0],[119.0, 36.0, 0],[119.0, 38.0, 0],[118.0, 39.0, 0],[118.0, 40.0, 0],[117.0, 41.0, 0],[117.0, 42.0, 0],[116.0, 43.0, 0],[116.0, 44.0, 0],[115.0, 45.0, 0],[115.0, 47.0, 0],[114.0, 48.0, 0],[114.0, 50.0, 0],[113.0, 51.0, 0],[113.0, 53.0, 0],[112.0, 54.0, 0],[112.0, 56.0, 0],[109.0, 59.0, 0],[102.0, 59.0, 0],[100.0, 57.0, 0],[100.0, 56.0, 0],[99.0, 55.0, 0],[99.0, 53.0, 0],[98.0, 52.0, 0],[98.0, 50.0, 0],[97.0, 49.0, 0],[97.0, 47.0, 0],[96.0, 46.0, 0],[96.0, 44.0, 0],[95.0, 43.0, 0],[95.0, 42.0, 0],[94.0, 41.0, 0],[94.0, 40.0, 0],[93.0, 39.0, 0],[93.0, 38.0, 0],[92.0, 37.0, 0],[92.0, 36.0, 0],[91.0, 35.0, 0],[91.0, 34.0, 0],[90.0, 33.0, 0],[90.0, 32.0, 0],[89.0, 31.0, 0],[89.0, 30.0, 0],[87.0, 28.0, 0],[87.0, 27.0, 0],[85.0, 25.0, 0],[85.0, 24.0, 0],[80.0, 19.0, 0],[80.0, 18.0, 0],[76.0, 14.0, 0],[75.0, 14.0, 0],[71.0, 10.0, 0],[70.0, 10.0, 0],[68.0, 8.0, 0],[67.0, 8.0, 0],[65.0, 6.0, 0],[64.0, 6.0, 0],[63.0, 5.0, 0],[62.0, 5.0, 0],[61.0, 4.0, 0],[60.0, 4.0, 0],[59.0, 3.0, 0],[58.0, 3.0, 0],[57.0, 2.0, 0],[55.0, 2.0, 0],[54.0, 1.0, 0],[51.0, 1.0, 0],[50.0, 0.0, 0],[37.0, 0.0, 0],[36.0, 1.0, 0],[34.0, 1.0, 0],[33.0, 2.0, 0],[31.0, 2.0, 0],[30.0, 3.0, 0],[29.0, 3.0, 0],[28.0, 4.0, 0],[27.0, 4.0, 0],[24.0, 7.0, 0],[23.0, 7.0, 0],[18.0, 12.0, 0],[18.0, 13.0, 0],[15.0, 16.0, 0],[15.0, 17.0, 0],[14.0, 18.0, 0],[14.0, 19.0, 0],[13.0, 20.0, 0],[13.0, 21.0, 0],[12.0, 22.0, 0],[12.0, 23.0, 0],[11.0, 24.0, 0],[11.0, 26.0, 0],[10.0, 27.0, 0],[10.0, 29.0, 0],[9.0, 30.0, 0],[9.0, 31.0, 0],[8.0, 32.0, 0],[8.0, 33.0, 0],[1.0, 40.0, 0],[1.0, 42.0, 0],[0.0, 43.0, 0]];
        VAR pos pos1{108} := [[118.0, 56.0, 0],[119.0, 55.0, 0],[119.0, 52.0, 0],[120.0, 51.0, 0],[120.0, 49.0, 0],[121.0, 48.0, 0],[121.0, 46.0, 0],[122.0, 45.0, 0],[122.0, 44.0, 0],[123.0, 43.0, 0],[123.0, 41.0, 0],[124.0, 40.0, 0],[124.0, 39.0, 0],[125.0, 38.0, 0],[125.0, 37.0, 0],[126.0, 36.0, 0],[126.0, 35.0, 0],[127.0, 34.0, 0],[127.0, 33.0, 0],[129.0, 31.0, 0],[129.0, 30.0, 0],[131.0, 28.0, 0],[131.0, 27.0, 0],[134.0, 24.0, 0],[134.0, 23.0, 0],[141.0, 16.0, 0],[142.0, 16.0, 0],[145.0, 13.0, 0],[146.0, 13.0, 0],[147.0, 12.0, 0],[148.0, 12.0, 0],[150.0, 10.0, 0],[152.0, 10.0, 0],[153.0, 9.0, 0],[154.0, 9.0, 0],[155.0, 8.0, 0],[157.0, 8.0, 0],[158.0, 7.0, 0],[160.0, 7.0, 0],[161.0, 6.0, 0],[175.0, 6.0, 0],[176.0, 7.0, 0],[178.0, 7.0, 0],[179.0, 8.0, 0],[180.0, 8.0, 0],[181.0, 9.0, 0],[182.0, 9.0, 0],[185.0, 12.0, 0],[186.0, 12.0, 0],[188.0, 14.0, 0],[188.0, 15.0, 0],[191.0, 18.0, 0],[191.0, 19.0, 0],[192.0, 20.0, 0],[192.0, 21.0, 0],[193.0, 22.0, 0],[193.0, 23.0, 0],[194.0, 24.0, 0],[194.0, 27.0, 0],[195.0, 28.0, 0],[195.0, 31.0, 0],[196.0, 32.0, 0],[196.0, 54.0, 0],[195.0, 55.0, 0],[195.0, 58.0, 0],[194.0, 59.0, 0],[194.0, 60.0, 0],[193.0, 61.0, 0],[193.0, 62.0, 0],[192.0, 63.0, 0],[192.0, 64.0, 0],[186.0, 70.0, 0],[185.0, 70.0, 0],[184.0, 71.0, 0],[183.0, 71.0, 0],[182.0, 72.0, 0],[181.0, 72.0, 0],[180.0, 73.0, 0],[178.0, 73.0, 0],[177.0, 74.0, 0],[174.0, 74.0, 0],[173.0, 75.0, 0],[169.0, 75.0, 0],[168.0, 76.0, 0],[163.0, 76.0, 0],[162.0, 77.0, 0],[156.0, 77.0, 0],[155.0, 78.0, 0],[152.0, 78.0, 0],[151.0, 77.0, 0],[147.0, 77.0, 0],[146.0, 76.0, 0],[141.0, 76.0, 0],[140.0, 75.0, 0],[136.0, 75.0, 0],[135.0, 74.0, 0],[132.0, 74.0, 0],[131.0, 73.0, 0],[129.0, 73.0, 0],[128.0, 72.0, 0],[126.0, 72.0, 0],[125.0, 71.0, 0],[124.0, 71.0, 0],[119.0, 66.0, 0],[119.0, 64.0, 0],[118.0, 63.0, 0],[118.0, 56.0, 0],[119.0, 55.0, 0]];
        VAR pos pos2{21} := [[156.0, 59.0, 0],[155.0, 60.0, 0],[155.0, 63.0, 0],[156.0, 64.0, 0],[156.0, 65.0, 0],[159.0, 68.0, 0],[165.0, 68.0, 0],[168.0, 65.0, 0],[168.0, 63.0, 0],[169.0, 62.0, 0],[169.0, 59.0, 0],[168.0, 58.0, 0],[167.0, 59.0, 0],[166.0, 59.0, 0],[163.0, 62.0, 0],[161.0, 62.0, 0],[160.0, 61.0, 0],[159.0, 61.0, 0],[157.0, 59.0, 0],[156.0, 59.0, 0],[155.0, 60.0, 0]];
        VAR pos pos3{19} := [[89.0, 77.0, 0],[92.0, 74.0, 0],[92.0, 73.0, 0],[94.0, 71.0, 0],[94.0, 70.0, 0],[98.0, 66.0, 0],[98.0, 65.0, 0],[99.0, 65.0, 0],[100.0, 64.0, 0],[107.0, 64.0, 0],[108.0, 65.0, 0],[111.0, 65.0, 0],[119.0, 73.0, 0],[119.0, 74.0, 0],[122.0, 77.0, 0],[122.0, 78.0, 0],[89.0, 78.0, 0],[89.0, 77.0, 0],[92.0, 74.0, 0]];
        VAR pos pos4{108} := [[14.0, 38.0, 0],[15.0, 37.0, 0],[15.0, 32.0, 0],[16.0, 31.0, 0],[16.0, 28.0, 0],[17.0, 27.0, 0],[17.0, 25.0, 0],[18.0, 24.0, 0],[18.0, 22.0, 0],[19.0, 21.0, 0],[19.0, 20.0, 0],[20.0, 19.0, 0],[20.0, 18.0, 0],[21.0, 17.0, 0],[21.0, 16.0, 0],[27.0, 10.0, 0],[28.0, 10.0, 0],[29.0, 9.0, 0],[30.0, 9.0, 0],[31.0, 8.0, 0],[33.0, 8.0, 0],[34.0, 7.0, 0],[36.0, 7.0, 0],[37.0, 6.0, 0],[50.0, 6.0, 0],[51.0, 7.0, 0],[53.0, 7.0, 0],[54.0, 8.0, 0],[55.0, 8.0, 0],[56.0, 9.0, 0],[58.0, 9.0, 0],[59.0, 10.0, 0],[60.0, 10.0, 0],[62.0, 12.0, 0],[63.0, 12.0, 0],[64.0, 13.0, 0],[65.0, 13.0, 0],[67.0, 15.0, 0],[68.0, 15.0, 0],[73.0, 20.0, 0],[74.0, 20.0, 0],[76.0, 22.0, 0],[76.0, 23.0, 0],[81.0, 28.0, 0],[81.0, 29.0, 0],[83.0, 31.0, 0],[83.0, 32.0, 0],[84.0, 33.0, 0],[84.0, 34.0, 0],[86.0, 36.0, 0],[86.0, 37.0, 0],[87.0, 38.0, 0],[87.0, 39.0, 0],[88.0, 40.0, 0],[88.0, 42.0, 0],[89.0, 43.0, 0],[89.0, 44.0, 0],[90.0, 45.0, 0],[90.0, 47.0, 0],[91.0, 48.0, 0],[91.0, 51.0, 0],[92.0, 52.0, 0],[92.0, 54.0, 0],[93.0, 55.0, 0],[93.0, 65.0, 0],[92.0, 66.0, 0],[92.0, 67.0, 0],[88.0, 71.0, 0],[87.0, 71.0, 0],[86.0, 72.0, 0],[84.0, 72.0, 0],[83.0, 73.0, 0],[81.0, 73.0, 0],[80.0, 74.0, 0],[77.0, 74.0, 0],[76.0, 75.0, 0],[72.0, 75.0, 0],[71.0, 76.0, 0],[67.0, 76.0, 0],[66.0, 77.0, 0],[61.0, 77.0, 0],[60.0, 78.0, 0],[57.0, 78.0, 0],[56.0, 77.0, 0],[48.0, 77.0, 0],[47.0, 76.0, 0],[40.0, 76.0, 0],[39.0, 75.0, 0],[35.0, 75.0, 0],[34.0, 74.0, 0],[32.0, 74.0, 0],[31.0, 73.0, 0],[29.0, 73.0, 0],[28.0, 72.0, 0],[27.0, 72.0, 0],[26.0, 71.0, 0],[25.0, 71.0, 0],[19.0, 65.0, 0],[19.0, 64.0, 0],[17.0, 62.0, 0],[17.0, 60.0, 0],[16.0, 59.0, 0],[16.0, 57.0, 0],[15.0, 56.0, 0],[15.0, 52.0, 0],[14.0, 51.0, 0],[14.0, 38.0, 0],[15.0, 37.0, 0]];
        VAR pos pos5{16} := [[40.0, 59.0, 0],[39.0, 60.0, 0],[39.0, 62.0, 0],[40.0, 63.0, 0],[40.0, 65.0, 0],[43.0, 68.0, 0],[44.0, 68.0, 0],[45.0, 67.0, 0],[47.0, 67.0, 0],[51.0, 63.0, 0],[51.0, 59.0, 0],[49.0, 57.0, 0],[46.0, 60.0, 0],[41.0, 60.0, 0],[40.0, 59.0, 0],[39.0, 60.0, 0]];

        ! Define variables to be used while drawing
        VAR pos position := [0,0,0];
        VAR robtarget next_target := [[0,0,0],[0,0,1,0],[0,0,0,0],[9E+09,9E+09,9E+09,9E+09,9E+09,9E+09]];

        ! Update the penup_offset based on the z_offset
        penup_offset := z_offset + penup_offset;

        ! Raise pen to avoid drawing of surface while moving to the new approach position
        position := pos0{1} * font_size;
        next_target.trans := position;
        MoveJ Offs(next_target, x_offset, y_offset, penup_offset),approach_speed,fine,Alex_Pen_ABB\WObj:=WorkSurface;

        ! Drop pen
        MoveL Offs(next_target, x_offset, y_offset, z_offset),approach_speed,fine,Alex_Pen_ABB\WObj:=WorkSurface;

        FOR index FROM 1 TO Dim(pos0, 1) DO
            position := pos0{index} * font_size;
            next_target.trans := position;

            MoveL Offs(next_target, x_offset, y_offset, z_offset),approach_speed,fine,Alex_Pen_ABB\WObj:=WorkSurface;
        ENDFOR

        ! Raise pen
        MoveL Offs(next_target, x_offset, y_offset, penup_offset),approach_speed,fine,Alex_Pen_ABB\WObj:=WorkSurface;

        ! Raise pen to avoid drawing of surface while moving to the new approach position
        position := pos1{1} * font_size;
        next_target.trans := position;
        MoveJ Offs(next_target, x_offset, y_offset, penup_offset),approach_speed,fine,Alex_Pen_ABB\WObj:=WorkSurface;

        ! Drop pen
        MoveL Offs(next_target, x_offset, y_offset, z_offset),approach_speed,fine,Alex_Pen_ABB\WObj:=WorkSurface;

        FOR index FROM 1 TO Dim(pos1, 1) DO
            position := pos1{index} * font_size;
            next_target.trans := position;

            MoveL Offs(next_target, x_offset, y_offset, z_offset),approach_speed,fine,Alex_Pen_ABB\WObj:=WorkSurface;
        ENDFOR

        ! Raise pen
        MoveL Offs(next_target, x_offset, y_offset, penup_offset),approach_speed,fine,Alex_Pen_ABB\WObj:=WorkSurface;

        ! Raise pen to avoid drawing of surface while moving to the new approach position
        position := pos2{1} * font_size;
        next_target.trans := position;
        MoveJ Offs(next_target, x_offset, y_offset, penup_offset),approach_speed,fine,Alex_Pen_ABB\WObj:=WorkSurface;

        ! Drop pen
        MoveL Offs(next_target, x_offset, y_offset, z_offset),approach_speed,fine,Alex_Pen_ABB\WObj:=WorkSurface;

        FOR index FROM 1 TO Dim(pos2, 1) DO
            position := pos2{index} * font_size;
            next_target.trans := position;

            MoveL Offs(next_target, x_offset, y_offset, z_offset),approach_speed,fine,Alex_Pen_ABB\WObj:=WorkSurface;
        ENDFOR

        ! Raise pen
        MoveL Offs(next_target, x_offset, y_offset, penup_offset),approach_speed,fine,Alex_Pen_ABB\WObj:=WorkSurface;

        ! Raise pen to avoid drawing of surface while moving to the new approach position
        position := pos3{1} * font_size;
        next_target.trans := position;
        MoveJ Offs(next_target, x_offset, y_offset, penup_offset),approach_speed,fine,Alex_Pen_ABB\WObj:=WorkSurface;

        ! Drop pen
        MoveL Offs(next_target, x_offset, y_offset, z_offset),approach_speed,fine,Alex_Pen_ABB\WObj:=WorkSurface;

        FOR index FROM 1 TO Dim(pos3, 1) DO
            position := pos3{index} * font_size;
            next_target.trans := position;

            MoveL Offs(next_target, x_offset, y_offset, z_offset),approach_speed,fine,Alex_Pen_ABB\WObj:=WorkSurface;
        ENDFOR

        ! Raise pen
        MoveL Offs(next_target, x_offset, y_offset, penup_offset),approach_speed,fine,Alex_Pen_ABB\WObj:=WorkSurface;

        ! Raise pen to avoid drawing of surface while moving to the new approach position
        position := pos4{1} * font_size;
        next_target.trans := position;
        MoveJ Offs(next_target, x_offset, y_offset, penup_offset),approach_speed,fine,Alex_Pen_ABB\WObj:=WorkSurface;

        ! Drop pen
        MoveL Offs(next_target, x_offset, y_offset, z_offset),approach_speed,fine,Alex_Pen_ABB\WObj:=WorkSurface;

        FOR index FROM 1 TO Dim(pos4, 1) DO
            position := pos4{index} * font_size;
            next_target.trans := position;

            MoveL Offs(next_target, x_offset, y_offset, z_offset),approach_speed,fine,Alex_Pen_ABB\WObj:=WorkSurface;
        ENDFOR

        ! Raise pen
        MoveL Offs(next_target, x_offset, y_offset, penup_offset),approach_speed,fine,Alex_Pen_ABB\WObj:=WorkSurface;

        ! Raise pen to avoid drawing of surface while moving to the new approach position
        position := pos5{1} * font_size;
        next_target.trans := position;
        MoveJ Offs(next_target, x_offset, y_offset, penup_offset),approach_speed,fine,Alex_Pen_ABB\WObj:=WorkSurface;

        ! Drop pen
        MoveL Offs(next_target, x_offset, y_offset, z_offset),approach_speed,fine,Alex_Pen_ABB\WObj:=WorkSurface;

        FOR index FROM 1 TO Dim(pos5, 1) DO
            position := pos5{index} * font_size;
            next_target.trans := position;

            MoveL Offs(next_target, x_offset, y_offset, z_offset),approach_speed,fine,Alex_Pen_ABB\WObj:=WorkSurface;
        ENDFOR

        ! Raise pen
        MoveL Offs(next_target, x_offset, y_offset, penup_offset),approach_speed,fine,Alex_Pen_ABB\WObj:=WorkSurface;

    ENDPROC

    !***********************************************************
    !
    ! Procedure DrawArtWork_Glasses
    !   This procedure draws the bottom border artwork on the work surface
    !   This is used by the Special User function
    !
    ! Example
    !   VAR speeddata approach_speed := v100;  // Approach speed for arm
    !   VAR speeddata write_speed := v80;      // Write speed for arm
    !   VAR num x_offset := 0;                 // x offset from worksurface origin
    !   VAR num y_offset := 0;                 // y offset from worksurface origin
    !   VAR num z_offset := 0;                 // z offset from worksurface origin
    !   VAR num pen_offset := 30;              // Defines pen position for pen up
    !
    !   DrawArtWork_ArtBorder 1.0, approach_speed, write_speed, x_offset, y_offset, z_offset, penup_offset;
    !
    !***********************************************************
    PROC DrawArtWork_ArtBorder(num font_size, speeddata approach_speed, speeddata write_speed, num x_offset, num y_offset, num z_offset, num penup_offset)
        ! Define all points for artwork
        VAR pos pos0{117} := [[494.0, 142.0, 0],[493.0, 143.0, 0],[493.0, 172.0, 0],[494.0, 173.0, 0],[497.0, 173.0, 0],[498.0, 174.0, 0],[509.0, 174.0, 0],[510.0, 175.0, 0],[522.0, 175.0, 0],[523.0, 176.0, 0],[534.0, 176.0, 0],[535.0, 177.0, 0],[543.0, 177.0, 0],[544.0, 176.0, 0],[555.0, 176.0, 0],[556.0, 175.0, 0],[567.0, 175.0, 0],[568.0, 174.0, 0],[579.0, 174.0, 0],[580.0, 173.0, 0],[583.0, 173.0, 0],[584.0, 172.0, 0],[584.0, 162.0, 0],[585.0, 161.0, 0],[585.0, 147.0, 0],[584.0, 146.0, 0],[584.0, 136.0, 0],[583.0, 135.0, 0],[583.0, 131.0, 0],[582.0, 130.0, 0],[582.0, 126.0, 0],[581.0, 125.0, 0],[581.0, 120.0, 0],[580.0, 119.0, 0],[580.0, 117.0, 0],[579.0, 116.0, 0],[579.0, 114.0, 0],[578.0, 113.0, 0],[578.0, 112.0, 0],[576.0, 110.0, 0],[576.0, 109.0, 0],[575.0, 108.0, 0],[575.0, 107.0, 0],[574.0, 106.0, 0],[574.0, 105.0, 0],[573.0, 104.0, 0],[573.0, 103.0, 0],[572.0, 102.0, 0],[572.0, 101.0, 0],[570.0, 99.0, 0],[570.0, 98.0, 0],[569.0, 97.0, 0],[569.0, 96.0, 0],[564.0, 91.0, 0],[564.0, 90.0, 0],[561.0, 87.0, 0],[560.0, 87.0, 0],[558.0, 85.0, 0],[558.0, 84.0, 0],[557.0, 83.0, 0],[556.0, 83.0, 0],[553.0, 80.0, 0],[552.0, 80.0, 0],[549.0, 77.0, 0],[548.0, 77.0, 0],[547.0, 76.0, 0],[546.0, 76.0, 0],[545.0, 75.0, 0],[544.0, 75.0, 0],[543.0, 74.0, 0],[542.0, 74.0, 0],[541.0, 73.0, 0],[540.0, 73.0, 0],[539.0, 72.0, 0],[538.0, 73.0, 0],[537.0, 73.0, 0],[536.0, 74.0, 0],[535.0, 74.0, 0],[533.0, 76.0, 0],[531.0, 76.0, 0],[530.0, 77.0, 0],[529.0, 77.0, 0],[527.0, 79.0, 0],[526.0, 79.0, 0],[518.0, 87.0, 0],[517.0, 87.0, 0],[511.0, 93.0, 0],[511.0, 94.0, 0],[510.0, 95.0, 0],[510.0, 96.0, 0],[509.0, 97.0, 0],[509.0, 98.0, 0],[506.0, 101.0, 0],[506.0, 102.0, 0],[504.0, 104.0, 0],[504.0, 105.0, 0],[503.0, 106.0, 0],[503.0, 107.0, 0],[502.0, 108.0, 0],[502.0, 109.0, 0],[501.0, 110.0, 0],[501.0, 111.0, 0],[500.0, 112.0, 0],[500.0, 113.0, 0],[499.0, 114.0, 0],[499.0, 118.0, 0],[498.0, 119.0, 0],[498.0, 121.0, 0],[497.0, 122.0, 0],[497.0, 124.0, 0],[496.0, 125.0, 0],[496.0, 129.0, 0],[495.0, 130.0, 0],[495.0, 134.0, 0],[494.0, 135.0, 0],[494.0, 142.0, 0],[493.0, 143.0, 0]];
        VAR pos pos1{60} := [[524.0, 162.0, 0],[525.0, 161.0, 0],[525.0, 160.0, 0],[526.0, 160.0, 0],[527.0, 159.0, 0],[527.0, 157.0, 0],[528.0, 156.0, 0],[528.0, 152.0, 0],[529.0, 151.0, 0],[529.0, 149.0, 0],[530.0, 149.0, 0],[531.0, 148.0, 0],[532.0, 148.0, 0],[533.0, 147.0, 0],[545.0, 147.0, 0],[546.0, 148.0, 0],[547.0, 148.0, 0],[549.0, 150.0, 0],[549.0, 154.0, 0],[550.0, 155.0, 0],[550.0, 158.0, 0],[552.0, 160.0, 0],[553.0, 160.0, 0],[553.0, 164.0, 0],[552.0, 165.0, 0],[551.0, 165.0, 0],[550.0, 164.0, 0],[550.0, 163.0, 0],[549.0, 162.0, 0],[549.0, 159.0, 0],[548.0, 158.0, 0],[547.0, 158.0, 0],[546.0, 157.0, 0],[545.0, 157.0, 0],[544.0, 158.0, 0],[541.0, 158.0, 0],[540.0, 159.0, 0],[540.0, 164.0, 0],[541.0, 165.0, 0],[540.0, 166.0, 0],[540.0, 168.0, 0],[537.0, 168.0, 0],[537.0, 166.0, 0],[536.0, 165.0, 0],[538.0, 163.0, 0],[538.0, 162.0, 0],[537.0, 161.0, 0],[537.0, 159.0, 0],[536.0, 158.0, 0],[534.0, 158.0, 0],[533.0, 157.0, 0],[531.0, 157.0, 0],[528.0, 160.0, 0],[528.0, 161.0, 0],[529.0, 162.0, 0],[526.0, 165.0, 0],[525.0, 164.0, 0],[524.0, 164.0, 0],[524.0, 162.0, 0],[525.0, 161.0, 0]];
        VAR pos pos2{17} := [[531.0, 149.0, 0],[530.0, 150.0, 0],[530.0, 151.0, 0],[531.0, 152.0, 0],[534.0, 152.0, 0],[535.0, 153.0, 0],[543.0, 153.0, 0],[544.0, 152.0, 0],[546.0, 152.0, 0],[548.0, 150.0, 0],[547.0, 149.0, 0],[546.0, 149.0, 0],[545.0, 148.0, 0],[533.0, 148.0, 0],[532.0, 149.0, 0],[531.0, 149.0, 0],[530.0, 150.0, 0]];
        VAR pos pos3{52} := [[519.0, 91.0, 0],[520.0, 90.0, 0],[521.0, 90.0, 0],[522.0, 91.0, 0],[523.0, 91.0, 0],[524.0, 92.0, 0],[525.0, 92.0, 0],[526.0, 93.0, 0],[527.0, 93.0, 0],[528.0, 92.0, 0],[526.0, 90.0, 0],[527.0, 89.0, 0],[528.0, 89.0, 0],[529.0, 90.0, 0],[529.0, 93.0, 0],[530.0, 94.0, 0],[533.0, 94.0, 0],[534.0, 95.0, 0],[540.0, 95.0, 0],[541.0, 94.0, 0],[543.0, 94.0, 0],[545.0, 96.0, 0],[546.0, 96.0, 0],[548.0, 94.0, 0],[548.0, 90.0, 0],[557.0, 90.0, 0],[557.0, 93.0, 0],[555.0, 95.0, 0],[554.0, 95.0, 0],[553.0, 96.0, 0],[552.0, 96.0, 0],[551.0, 97.0, 0],[549.0, 97.0, 0],[548.0, 98.0, 0],[546.0, 98.0, 0],[545.0, 99.0, 0],[535.0, 99.0, 0],[534.0, 98.0, 0],[531.0, 98.0, 0],[530.0, 97.0, 0],[528.0, 97.0, 0],[527.0, 98.0, 0],[528.0, 99.0, 0],[526.0, 99.0, 0],[526.0, 97.0, 0],[524.0, 95.0, 0],[523.0, 95.0, 0],[521.0, 93.0, 0],[520.0, 93.0, 0],[519.0, 92.0, 0],[519.0, 91.0, 0],[520.0, 90.0, 0]];
        VAR pos pos4{66} := [[512.0, 107.0, 0],[513.0, 106.0, 0],[513.0, 105.0, 0],[515.0, 105.0, 0],[516.0, 106.0, 0],[517.0, 106.0, 0],[518.0, 107.0, 0],[520.0, 107.0, 0],[521.0, 108.0, 0],[522.0, 108.0, 0],[523.0, 107.0, 0],[523.0, 105.0, 0],[524.0, 105.0, 0],[525.0, 106.0, 0],[525.0, 109.0, 0],[526.0, 110.0, 0],[527.0, 110.0, 0],[528.0, 111.0, 0],[534.0, 111.0, 0],[535.0, 112.0, 0],[537.0, 112.0, 0],[538.0, 111.0, 0],[543.0, 111.0, 0],[544.0, 110.0, 0],[545.0, 110.0, 0],[545.0, 111.0, 0],[546.0, 112.0, 0],[550.0, 112.0, 0],[551.0, 111.0, 0],[551.0, 106.0, 0],[552.0, 105.0, 0],[564.0, 105.0, 0],[564.0, 107.0, 0],[560.0, 111.0, 0],[558.0, 111.0, 0],[556.0, 113.0, 0],[555.0, 113.0, 0],[554.0, 114.0, 0],[552.0, 114.0, 0],[551.0, 115.0, 0],[547.0, 115.0, 0],[546.0, 116.0, 0],[535.0, 116.0, 0],[534.0, 115.0, 0],[531.0, 115.0, 0],[530.0, 114.0, 0],[527.0, 114.0, 0],[526.0, 113.0, 0],[524.0, 113.0, 0],[523.0, 114.0, 0],[523.0, 115.0, 0],[524.0, 116.0, 0],[524.0, 117.0, 0],[523.0, 117.0, 0],[523.0, 116.0, 0],[522.0, 115.0, 0],[522.0, 112.0, 0],[521.0, 111.0, 0],[518.0, 111.0, 0],[517.0, 110.0, 0],[515.0, 110.0, 0],[514.0, 109.0, 0],[513.0, 109.0, 0],[512.0, 108.0, 0],[512.0, 107.0, 0],[513.0, 106.0, 0]];
        VAR pos pos5{6} := [[523.0, 107.0, 0],[522.0, 108.0, 0],[523.0, 109.0, 0],[524.0, 108.0, 0],[523.0, 107.0, 0],[522.0, 108.0, 0]];
        VAR pos pos6{74} := [[507.0, 125.0, 0],[508.0, 124.0, 0],[512.0, 124.0, 0],[513.0, 125.0, 0],[515.0, 125.0, 0],[516.0, 126.0, 0],[518.0, 126.0, 0],[519.0, 127.0, 0],[520.0, 127.0, 0],[521.0, 126.0, 0],[521.0, 125.0, 0],[519.0, 123.0, 0],[522.0, 123.0, 0],[522.0, 128.0, 0],[523.0, 129.0, 0],[526.0, 129.0, 0],[527.0, 130.0, 0],[541.0, 130.0, 0],[542.0, 129.0, 0],[545.0, 129.0, 0],[546.0, 128.0, 0],[547.0, 128.0, 0],[549.0, 130.0, 0],[550.0, 130.0, 0],[551.0, 131.0, 0],[552.0, 131.0, 0],[555.0, 128.0, 0],[555.0, 125.0, 0],[554.0, 124.0, 0],[555.0, 124.0, 0],[557.0, 122.0, 0],[558.0, 123.0, 0],[559.0, 122.0, 0],[569.0, 122.0, 0],[570.0, 123.0, 0],[569.0, 124.0, 0],[569.0, 126.0, 0],[564.0, 131.0, 0],[563.0, 131.0, 0],[562.0, 132.0, 0],[561.0, 132.0, 0],[560.0, 133.0, 0],[559.0, 133.0, 0],[558.0, 134.0, 0],[557.0, 134.0, 0],[556.0, 135.0, 0],[548.0, 135.0, 0],[547.0, 136.0, 0],[534.0, 136.0, 0],[533.0, 135.0, 0],[526.0, 135.0, 0],[525.0, 134.0, 0],[523.0, 134.0, 0],[522.0, 133.0, 0],[521.0, 133.0, 0],[520.0, 134.0, 0],[520.0, 135.0, 0],[521.0, 136.0, 0],[522.0, 136.0, 0],[521.0, 137.0, 0],[520.0, 137.0, 0],[518.0, 135.0, 0],[518.0, 132.0, 0],[517.0, 131.0, 0],[515.0, 131.0, 0],[514.0, 130.0, 0],[513.0, 130.0, 0],[511.0, 128.0, 0],[510.0, 128.0, 0],[509.0, 127.0, 0],[508.0, 127.0, 0],[507.0, 126.0, 0],[507.0, 125.0, 0],[508.0, 124.0, 0]];
        VAR pos pos7{36} := [[226.0, 120.0, 0],[225.0, 121.0, 0],[225.0, 163.0, 0],[226.0, 164.0, 0],[238.0, 164.0, 0],[239.0, 163.0, 0],[241.0, 163.0, 0],[242.0, 162.0, 0],[243.0, 162.0, 0],[245.0, 160.0, 0],[246.0, 160.0, 0],[250.0, 156.0, 0],[250.0, 155.0, 0],[252.0, 153.0, 0],[252.0, 151.0, 0],[253.0, 150.0, 0],[253.0, 148.0, 0],[254.0, 147.0, 0],[254.0, 140.0, 0],[253.0, 139.0, 0],[253.0, 137.0, 0],[252.0, 136.0, 0],[252.0, 134.0, 0],[250.0, 132.0, 0],[250.0, 131.0, 0],[246.0, 127.0, 0],[245.0, 127.0, 0],[244.0, 126.0, 0],[245.0, 125.0, 0],[246.0, 125.0, 0],[247.0, 124.0, 0],[248.0, 124.0, 0],[251.0, 121.0, 0],[250.0, 120.0, 0],[226.0, 120.0, 0],[225.0, 121.0, 0]];
        VAR pos pos8{34} := [[226.0, 73.0, 0],[225.0, 74.0, 0],[225.0, 116.0, 0],[226.0, 117.0, 0],[255.0, 117.0, 0],[256.0, 116.0, 0],[256.0, 115.0, 0],[257.0, 114.0, 0],[257.0, 113.0, 0],[259.0, 111.0, 0],[259.0, 109.0, 0],[260.0, 108.0, 0],[260.0, 104.0, 0],[261.0, 103.0, 0],[261.0, 98.0, 0],[260.0, 97.0, 0],[260.0, 93.0, 0],[259.0, 92.0, 0],[259.0, 90.0, 0],[258.0, 89.0, 0],[258.0, 88.0, 0],[256.0, 86.0, 0],[256.0, 85.0, 0],[248.0, 77.0, 0],[247.0, 77.0, 0],[246.0, 76.0, 0],[245.0, 76.0, 0],[244.0, 75.0, 0],[243.0, 75.0, 0],[242.0, 74.0, 0],[240.0, 74.0, 0],[239.0, 73.0, 0],[226.0, 73.0, 0],[225.0, 74.0, 0]];
        VAR pos pos9{10} := [[197.0, 120.0, 0],[196.0, 121.0, 0],[196.0, 163.0, 0],[197.0, 164.0, 0],[222.0, 164.0, 0],[223.0, 163.0, 0],[223.0, 122.0, 0],[221.0, 120.0, 0],[197.0, 120.0, 0],[196.0, 121.0, 0]];
        VAR pos pos10{10} := [[197.0, 73.0, 0],[196.0, 74.0, 0],[196.0, 116.0, 0],[197.0, 117.0, 0],[222.0, 117.0, 0],[223.0, 116.0, 0],[223.0, 74.0, 0],[222.0, 73.0, 0],[197.0, 73.0, 0],[196.0, 74.0, 0]];
        VAR pos pos11{37} := [[155.0, 120.0, 0],[154.0, 121.0, 0],[154.0, 163.0, 0],[155.0, 164.0, 0],[168.0, 164.0, 0],[169.0, 163.0, 0],[170.0, 163.0, 0],[171.0, 162.0, 0],[172.0, 162.0, 0],[173.0, 161.0, 0],[174.0, 161.0, 0],[180.0, 155.0, 0],[180.0, 154.0, 0],[181.0, 153.0, 0],[181.0, 152.0, 0],[182.0, 151.0, 0],[182.0, 149.0, 0],[183.0, 148.0, 0],[183.0, 139.0, 0],[182.0, 138.0, 0],[182.0, 136.0, 0],[181.0, 135.0, 0],[181.0, 134.0, 0],[180.0, 133.0, 0],[180.0, 132.0, 0],[174.0, 126.0, 0],[173.0, 126.0, 0],[174.0, 125.0, 0],[175.0, 125.0, 0],[176.0, 124.0, 0],[177.0, 124.0, 0],[179.0, 122.0, 0],[180.0, 122.0, 0],[181.0, 121.0, 0],[180.0, 120.0, 0],[155.0, 120.0, 0],[154.0, 121.0, 0]];
        VAR pos pos12{38} := [[155.0, 73.0, 0],[154.0, 74.0, 0],[154.0, 116.0, 0],[155.0, 117.0, 0],[184.0, 117.0, 0],[186.0, 115.0, 0],[186.0, 114.0, 0],[187.0, 113.0, 0],[187.0, 112.0, 0],[188.0, 111.0, 0],[188.0, 110.0, 0],[189.0, 109.0, 0],[189.0, 106.0, 0],[190.0, 105.0, 0],[190.0, 96.0, 0],[189.0, 95.0, 0],[189.0, 92.0, 0],[188.0, 91.0, 0],[188.0, 90.0, 0],[187.0, 89.0, 0],[187.0, 88.0, 0],[186.0, 87.0, 0],[186.0, 86.0, 0],[184.0, 84.0, 0],[184.0, 83.0, 0],[180.0, 79.0, 0],[179.0, 79.0, 0],[177.0, 77.0, 0],[176.0, 77.0, 0],[175.0, 76.0, 0],[174.0, 76.0, 0],[173.0, 75.0, 0],[172.0, 75.0, 0],[171.0, 74.0, 0],[169.0, 74.0, 0],[168.0, 73.0, 0],[155.0, 73.0, 0],[154.0, 74.0, 0]];
        VAR pos pos13{10} := [[127.0, 120.0, 0],[126.0, 121.0, 0],[126.0, 163.0, 0],[127.0, 164.0, 0],[151.0, 164.0, 0],[152.0, 163.0, 0],[152.0, 121.0, 0],[151.0, 120.0, 0],[127.0, 120.0, 0],[126.0, 121.0, 0]];
        VAR pos pos14{10} := [[127.0, 73.0, 0],[126.0, 74.0, 0],[126.0, 116.0, 0],[127.0, 117.0, 0],[151.0, 117.0, 0],[152.0, 116.0, 0],[152.0, 74.0, 0],[151.0, 73.0, 0],[127.0, 73.0, 0],[126.0, 74.0, 0]];
        VAR pos pos15{38} := [[77.0, 120.0, 0],[76.0, 121.0, 0],[76.0, 163.0, 0],[77.0, 164.0, 0],[88.0, 164.0, 0],[89.0, 163.0, 0],[89.0, 161.0, 0],[90.0, 160.0, 0],[90.0, 158.0, 0],[91.0, 157.0, 0],[91.0, 156.0, 0],[92.0, 155.0, 0],[92.0, 153.0, 0],[93.0, 152.0, 0],[93.0, 150.0, 0],[94.0, 149.0, 0],[94.0, 147.0, 0],[95.0, 146.0, 0],[95.0, 144.0, 0],[96.0, 143.0, 0],[96.0, 141.0, 0],[97.0, 140.0, 0],[97.0, 138.0, 0],[98.0, 137.0, 0],[98.0, 135.0, 0],[99.0, 134.0, 0],[99.0, 133.0, 0],[100.0, 132.0, 0],[100.0, 130.0, 0],[101.0, 129.0, 0],[101.0, 127.0, 0],[102.0, 126.0, 0],[102.0, 124.0, 0],[103.0, 123.0, 0],[103.0, 121.0, 0],[102.0, 120.0, 0],[77.0, 120.0, 0],[76.0, 121.0, 0]];
        VAR pos pos16{52} := [[77.0, 91.0, 0],[76.0, 92.0, 0],[76.0, 116.0, 0],[77.0, 117.0, 0],[104.0, 117.0, 0],[106.0, 115.0, 0],[106.0, 113.0, 0],[107.0, 112.0, 0],[107.0, 110.0, 0],[108.0, 109.0, 0],[108.0, 107.0, 0],[109.0, 106.0, 0],[109.0, 104.0, 0],[110.0, 103.0, 0],[110.0, 101.0, 0],[111.0, 100.0, 0],[111.0, 99.0, 0],[112.0, 98.0, 0],[112.0, 96.0, 0],[113.0, 95.0, 0],[113.0, 93.0, 0],[114.0, 92.0, 0],[114.0, 90.0, 0],[115.0, 89.0, 0],[115.0, 87.0, 0],[116.0, 86.0, 0],[116.0, 84.0, 0],[117.0, 83.0, 0],[117.0, 81.0, 0],[118.0, 80.0, 0],[118.0, 79.0, 0],[119.0, 78.0, 0],[119.0, 76.0, 0],[120.0, 75.0, 0],[120.0, 74.0, 0],[119.0, 73.0, 0],[97.0, 73.0, 0],[96.0, 74.0, 0],[96.0, 76.0, 0],[95.0, 77.0, 0],[95.0, 79.0, 0],[94.0, 80.0, 0],[94.0, 81.0, 0],[93.0, 82.0, 0],[93.0, 84.0, 0],[92.0, 85.0, 0],[92.0, 87.0, 0],[91.0, 88.0, 0],[91.0, 90.0, 0],[90.0, 91.0, 0],[77.0, 91.0, 0],[76.0, 92.0, 0]];
        VAR pos pos17{39} := [[46.0, 120.0, 0],[45.0, 121.0, 0],[46.0, 122.0, 0],[46.0, 124.0, 0],[47.0, 125.0, 0],[47.0, 127.0, 0],[48.0, 128.0, 0],[48.0, 130.0, 0],[49.0, 131.0, 0],[49.0, 133.0, 0],[50.0, 134.0, 0],[50.0, 135.0, 0],[51.0, 136.0, 0],[51.0, 139.0, 0],[52.0, 140.0, 0],[52.0, 141.0, 0],[53.0, 142.0, 0],[53.0, 144.0, 0],[54.0, 145.0, 0],[54.0, 147.0, 0],[55.0, 148.0, 0],[55.0, 150.0, 0],[56.0, 151.0, 0],[56.0, 153.0, 0],[57.0, 154.0, 0],[57.0, 156.0, 0],[58.0, 157.0, 0],[58.0, 159.0, 0],[59.0, 160.0, 0],[59.0, 161.0, 0],[60.0, 162.0, 0],[60.0, 163.0, 0],[61.0, 164.0, 0],[72.0, 164.0, 0],[73.0, 163.0, 0],[73.0, 121.0, 0],[72.0, 120.0, 0],[46.0, 120.0, 0],[45.0, 121.0, 0]];
        VAR pos pos18{51} := [[30.0, 73.0, 0],[29.0, 74.0, 0],[29.0, 76.0, 0],[30.0, 77.0, 0],[30.0, 79.0, 0],[31.0, 80.0, 0],[31.0, 81.0, 0],[32.0, 82.0, 0],[32.0, 84.0, 0],[33.0, 85.0, 0],[33.0, 87.0, 0],[34.0, 88.0, 0],[34.0, 90.0, 0],[35.0, 91.0, 0],[35.0, 93.0, 0],[36.0, 94.0, 0],[36.0, 95.0, 0],[37.0, 96.0, 0],[37.0, 99.0, 0],[38.0, 100.0, 0],[38.0, 101.0, 0],[39.0, 102.0, 0],[39.0, 104.0, 0],[40.0, 105.0, 0],[40.0, 107.0, 0],[41.0, 108.0, 0],[41.0, 110.0, 0],[42.0, 111.0, 0],[42.0, 113.0, 0],[43.0, 114.0, 0],[43.0, 116.0, 0],[44.0, 117.0, 0],[72.0, 117.0, 0],[73.0, 116.0, 0],[73.0, 92.0, 0],[72.0, 91.0, 0],[58.0, 91.0, 0],[58.0, 89.0, 0],[57.0, 88.0, 0],[57.0, 86.0, 0],[56.0, 85.0, 0],[56.0, 83.0, 0],[55.0, 82.0, 0],[55.0, 81.0, 0],[54.0, 80.0, 0],[54.0, 78.0, 0],[53.0, 77.0, 0],[53.0, 75.0, 0],[51.0, 73.0, 0],[30.0, 73.0, 0],[29.0, 74.0, 0]];

        ! Define variables to be used while drawing
        VAR pos position := [0,0,0];
        VAR robtarget next_target := [[0,0,0],[0,0,1,0],[0,0,0,0],[9E+09,9E+09,9E+09,9E+09,9E+09,9E+09]];

        ! Update the penup_offset based on the z_offset
        penup_offset := z_offset + penup_offset;

        ! Raise pen to avoid drawing of surface while moving to the new approach position
        position := pos0{1} * font_size;
        next_target.trans := position;
        MoveJ Offs(next_target, x_offset, y_offset, penup_offset),approach_speed,fine,Alex_Pen_ABB\WObj:=WorkSurface;

        ! Drop pen
        MoveL Offs(next_target, x_offset, y_offset, z_offset),approach_speed,fine,Alex_Pen_ABB\WObj:=WorkSurface;

        FOR index FROM 1 TO Dim(pos0, 1) DO
            position := pos0{index} * font_size;
            next_target.trans := position;

            MoveL Offs(next_target, x_offset, y_offset, z_offset),approach_speed,fine,Alex_Pen_ABB\WObj:=WorkSurface;
        ENDFOR

        ! Raise pen
        MoveL Offs(next_target, x_offset, y_offset, penup_offset),approach_speed,fine,Alex_Pen_ABB\WObj:=WorkSurface;

        ! Raise pen to avoid drawing of surface while moving to the new approach position
        position := pos1{1} * font_size;
        next_target.trans := position;
        MoveJ Offs(next_target, x_offset, y_offset, penup_offset),approach_speed,fine,Alex_Pen_ABB\WObj:=WorkSurface;

        ! Drop pen
        MoveL Offs(next_target, x_offset, y_offset, z_offset),approach_speed,fine,Alex_Pen_ABB\WObj:=WorkSurface;

        FOR index FROM 1 TO Dim(pos1, 1) DO
            position := pos1{index} * font_size;
            next_target.trans := position;

            MoveL Offs(next_target, x_offset, y_offset, z_offset),approach_speed,fine,Alex_Pen_ABB\WObj:=WorkSurface;
        ENDFOR

        ! Raise pen
        MoveL Offs(next_target, x_offset, y_offset, penup_offset),approach_speed,fine,Alex_Pen_ABB\WObj:=WorkSurface;

        ! Raise pen to avoid drawing of surface while moving to the new approach position
        position := pos2{1} * font_size;
        next_target.trans := position;
        MoveJ Offs(next_target, x_offset, y_offset, penup_offset),approach_speed,fine,Alex_Pen_ABB\WObj:=WorkSurface;

        ! Drop pen
        MoveL Offs(next_target, x_offset, y_offset, z_offset),approach_speed,fine,Alex_Pen_ABB\WObj:=WorkSurface;

        FOR index FROM 1 TO Dim(pos2, 1) DO
            position := pos2{index} * font_size;
            next_target.trans := position;

            MoveL Offs(next_target, x_offset, y_offset, z_offset),approach_speed,fine,Alex_Pen_ABB\WObj:=WorkSurface;
        ENDFOR

        ! Raise pen
        MoveL Offs(next_target, x_offset, y_offset, penup_offset),approach_speed,fine,Alex_Pen_ABB\WObj:=WorkSurface;

        ! Raise pen to avoid drawing of surface while moving to the new approach position
        position := pos3{1} * font_size;
        next_target.trans := position;
        MoveJ Offs(next_target, x_offset, y_offset, penup_offset),approach_speed,fine,Alex_Pen_ABB\WObj:=WorkSurface;

        ! Drop pen
        MoveL Offs(next_target, x_offset, y_offset, z_offset),approach_speed,fine,Alex_Pen_ABB\WObj:=WorkSurface;

        FOR index FROM 1 TO Dim(pos3, 1) DO
            position := pos3{index} * font_size;
            next_target.trans := position;

            MoveL Offs(next_target, x_offset, y_offset, z_offset),approach_speed,fine,Alex_Pen_ABB\WObj:=WorkSurface;
        ENDFOR

        ! Raise pen
        MoveL Offs(next_target, x_offset, y_offset, penup_offset),approach_speed,fine,Alex_Pen_ABB\WObj:=WorkSurface;

        ! Raise pen to avoid drawing of surface while moving to the new approach position
        position := pos4{1} * font_size;
        next_target.trans := position;
        MoveJ Offs(next_target, x_offset, y_offset, penup_offset),approach_speed,fine,Alex_Pen_ABB\WObj:=WorkSurface;

        ! Drop pen
        MoveL Offs(next_target, x_offset, y_offset, z_offset),approach_speed,fine,Alex_Pen_ABB\WObj:=WorkSurface;

        FOR index FROM 1 TO Dim(pos4, 1) DO
            position := pos4{index} * font_size;
            next_target.trans := position;

            MoveL Offs(next_target, x_offset, y_offset, z_offset),approach_speed,fine,Alex_Pen_ABB\WObj:=WorkSurface;
        ENDFOR

        ! Raise pen
        MoveL Offs(next_target, x_offset, y_offset, penup_offset),approach_speed,fine,Alex_Pen_ABB\WObj:=WorkSurface;

        ! Raise pen to avoid drawing of surface while moving to the new approach position
        position := pos5{1} * font_size;
        next_target.trans := position;
        MoveJ Offs(next_target, x_offset, y_offset, penup_offset),approach_speed,fine,Alex_Pen_ABB\WObj:=WorkSurface;

        ! Drop pen
        MoveL Offs(next_target, x_offset, y_offset, z_offset),approach_speed,fine,Alex_Pen_ABB\WObj:=WorkSurface;

        FOR index FROM 1 TO Dim(pos5, 1) DO
            position := pos5{index} * font_size;
            next_target.trans := position;

            MoveL Offs(next_target, x_offset, y_offset, z_offset),approach_speed,fine,Alex_Pen_ABB\WObj:=WorkSurface;
        ENDFOR

        ! Raise pen
        MoveL Offs(next_target, x_offset, y_offset, penup_offset),approach_speed,fine,Alex_Pen_ABB\WObj:=WorkSurface;

        ! Raise pen to avoid drawing of surface while moving to the new approach position
        position := pos6{1} * font_size;
        next_target.trans := position;
        MoveJ Offs(next_target, x_offset, y_offset, penup_offset),approach_speed,fine,Alex_Pen_ABB\WObj:=WorkSurface;

        ! Drop pen
        MoveL Offs(next_target, x_offset, y_offset, z_offset),approach_speed,fine,Alex_Pen_ABB\WObj:=WorkSurface;

        FOR index FROM 1 TO Dim(pos6, 1) DO
            position := pos6{index} * font_size;
            next_target.trans := position;

            MoveL Offs(next_target, x_offset, y_offset, z_offset),approach_speed,fine,Alex_Pen_ABB\WObj:=WorkSurface;
        ENDFOR

        ! Raise pen
        MoveL Offs(next_target, x_offset, y_offset, penup_offset),approach_speed,fine,Alex_Pen_ABB\WObj:=WorkSurface;

        ! Raise pen to avoid drawing of surface while moving to the new approach position
        position := pos7{1} * font_size;
        next_target.trans := position;
        MoveJ Offs(next_target, x_offset, y_offset, penup_offset),approach_speed,fine,Alex_Pen_ABB\WObj:=WorkSurface;

        ! Drop pen
        MoveL Offs(next_target, x_offset, y_offset, z_offset),approach_speed,fine,Alex_Pen_ABB\WObj:=WorkSurface;

        FOR index FROM 1 TO Dim(pos7, 1) DO
            position := pos7{index} * font_size;
            next_target.trans := position;

            MoveL Offs(next_target, x_offset, y_offset, z_offset),approach_speed,fine,Alex_Pen_ABB\WObj:=WorkSurface;
        ENDFOR

        ! Raise pen
        MoveL Offs(next_target, x_offset, y_offset, penup_offset),approach_speed,fine,Alex_Pen_ABB\WObj:=WorkSurface;

        ! Raise pen to avoid drawing of surface while moving to the new approach position
        position := pos8{1} * font_size;
        next_target.trans := position;
        MoveJ Offs(next_target, x_offset, y_offset, penup_offset),approach_speed,fine,Alex_Pen_ABB\WObj:=WorkSurface;

        ! Drop pen
        MoveL Offs(next_target, x_offset, y_offset, z_offset),approach_speed,fine,Alex_Pen_ABB\WObj:=WorkSurface;

        FOR index FROM 1 TO Dim(pos8, 1) DO
            position := pos8{index} * font_size;
            next_target.trans := position;

            MoveL Offs(next_target, x_offset, y_offset, z_offset),approach_speed,fine,Alex_Pen_ABB\WObj:=WorkSurface;
        ENDFOR

        ! Raise pen
        MoveL Offs(next_target, x_offset, y_offset, penup_offset),approach_speed,fine,Alex_Pen_ABB\WObj:=WorkSurface;

        ! Raise pen to avoid drawing of surface while moving to the new approach position
        position := pos9{1} * font_size;
        next_target.trans := position;
        MoveJ Offs(next_target, x_offset, y_offset, penup_offset),approach_speed,fine,Alex_Pen_ABB\WObj:=WorkSurface;

        ! Drop pen
        MoveL Offs(next_target, x_offset, y_offset, z_offset),approach_speed,fine,Alex_Pen_ABB\WObj:=WorkSurface;

        FOR index FROM 1 TO Dim(pos9, 1) DO
            position := pos9{index} * font_size;
            next_target.trans := position;

            MoveL Offs(next_target, x_offset, y_offset, z_offset),approach_speed,fine,Alex_Pen_ABB\WObj:=WorkSurface;
        ENDFOR

        ! Raise pen
        MoveL Offs(next_target, x_offset, y_offset, penup_offset),approach_speed,fine,Alex_Pen_ABB\WObj:=WorkSurface;

        ! Raise pen to avoid drawing of surface while moving to the new approach position
        position := pos10{1} * font_size;
        next_target.trans := position;
        MoveJ Offs(next_target, x_offset, y_offset, penup_offset),approach_speed,fine,Alex_Pen_ABB\WObj:=WorkSurface;

        ! Drop pen
        MoveL Offs(next_target, x_offset, y_offset, z_offset),approach_speed,fine,Alex_Pen_ABB\WObj:=WorkSurface;

        FOR index FROM 1 TO Dim(pos10, 1) DO
            position := pos10{index} * font_size;
            next_target.trans := position;

            MoveL Offs(next_target, x_offset, y_offset, z_offset),approach_speed,fine,Alex_Pen_ABB\WObj:=WorkSurface;
        ENDFOR

        ! Raise pen
        MoveL Offs(next_target, x_offset, y_offset, penup_offset),approach_speed,fine,Alex_Pen_ABB\WObj:=WorkSurface;

        ! Raise pen to avoid drawing of surface while moving to the new approach position
        position := pos11{1} * font_size;
        next_target.trans := position;
        MoveJ Offs(next_target, x_offset, y_offset, penup_offset),approach_speed,fine,Alex_Pen_ABB\WObj:=WorkSurface;

        ! Drop pen
        MoveL Offs(next_target, x_offset, y_offset, z_offset),approach_speed,fine,Alex_Pen_ABB\WObj:=WorkSurface;

        FOR index FROM 1 TO Dim(pos11, 1) DO
            position := pos11{index} * font_size;
            next_target.trans := position;

            MoveL Offs(next_target, x_offset, y_offset, z_offset),approach_speed,fine,Alex_Pen_ABB\WObj:=WorkSurface;
        ENDFOR

        ! Raise pen
        MoveL Offs(next_target, x_offset, y_offset, penup_offset),approach_speed,fine,Alex_Pen_ABB\WObj:=WorkSurface;

        ! Raise pen to avoid drawing of surface while moving to the new approach position
        position := pos12{1} * font_size;
        next_target.trans := position;
        MoveJ Offs(next_target, x_offset, y_offset, penup_offset),approach_speed,fine,Alex_Pen_ABB\WObj:=WorkSurface;

        ! Drop pen
        MoveL Offs(next_target, x_offset, y_offset, z_offset),approach_speed,fine,Alex_Pen_ABB\WObj:=WorkSurface;

        FOR index FROM 1 TO Dim(pos12, 1) DO
            position := pos12{index} * font_size;
            next_target.trans := position;

            MoveL Offs(next_target, x_offset, y_offset, z_offset),approach_speed,fine,Alex_Pen_ABB\WObj:=WorkSurface;
        ENDFOR

        ! Raise pen
        MoveL Offs(next_target, x_offset, y_offset, penup_offset),approach_speed,fine,Alex_Pen_ABB\WObj:=WorkSurface;

        ! Raise pen to avoid drawing of surface while moving to the new approach position
        position := pos13{1} * font_size;
        next_target.trans := position;
        MoveJ Offs(next_target, x_offset, y_offset, penup_offset),approach_speed,fine,Alex_Pen_ABB\WObj:=WorkSurface;

        ! Drop pen
        MoveL Offs(next_target, x_offset, y_offset, z_offset),approach_speed,fine,Alex_Pen_ABB\WObj:=WorkSurface;

        FOR index FROM 1 TO Dim(pos13, 1) DO
            position := pos13{index} * font_size;
            next_target.trans := position;

            MoveL Offs(next_target, x_offset, y_offset, z_offset),approach_speed,fine,Alex_Pen_ABB\WObj:=WorkSurface;
        ENDFOR

        ! Raise pen
        MoveL Offs(next_target, x_offset, y_offset, penup_offset),approach_speed,fine,Alex_Pen_ABB\WObj:=WorkSurface;

        ! Raise pen to avoid drawing of surface while moving to the new approach position
        position := pos14{1} * font_size;
        next_target.trans := position;
        MoveJ Offs(next_target, x_offset, y_offset, penup_offset),approach_speed,fine,Alex_Pen_ABB\WObj:=WorkSurface;

        ! Drop pen
        MoveL Offs(next_target, x_offset, y_offset, z_offset),approach_speed,fine,Alex_Pen_ABB\WObj:=WorkSurface;

        FOR index FROM 1 TO Dim(pos14, 1) DO
            position := pos14{index} * font_size;
            next_target.trans := position;

            MoveL Offs(next_target, x_offset, y_offset, z_offset),approach_speed,fine,Alex_Pen_ABB\WObj:=WorkSurface;
        ENDFOR

        ! Raise pen
        MoveL Offs(next_target, x_offset, y_offset, penup_offset),approach_speed,fine,Alex_Pen_ABB\WObj:=WorkSurface;

        ! Raise pen to avoid drawing of surface while moving to the new approach position
        position := pos15{1} * font_size;
        next_target.trans := position;
        MoveJ Offs(next_target, x_offset, y_offset, penup_offset),approach_speed,fine,Alex_Pen_ABB\WObj:=WorkSurface;

        ! Drop pen
        MoveL Offs(next_target, x_offset, y_offset, z_offset),approach_speed,fine,Alex_Pen_ABB\WObj:=WorkSurface;

        FOR index FROM 1 TO Dim(pos15, 1) DO
            position := pos15{index} * font_size;
            next_target.trans := position;

            MoveL Offs(next_target, x_offset, y_offset, z_offset),approach_speed,fine,Alex_Pen_ABB\WObj:=WorkSurface;
        ENDFOR

        ! Raise pen
        MoveL Offs(next_target, x_offset, y_offset, penup_offset),approach_speed,fine,Alex_Pen_ABB\WObj:=WorkSurface;

        ! Raise pen to avoid drawing of surface while moving to the new approach position
        position := pos16{1} * font_size;
        next_target.trans := position;
        MoveJ Offs(next_target, x_offset, y_offset, penup_offset),approach_speed,fine,Alex_Pen_ABB\WObj:=WorkSurface;

        ! Drop pen
        MoveL Offs(next_target, x_offset, y_offset, z_offset),approach_speed,fine,Alex_Pen_ABB\WObj:=WorkSurface;

        FOR index FROM 1 TO Dim(pos16, 1) DO
            position := pos16{index} * font_size;
            next_target.trans := position;

            MoveL Offs(next_target, x_offset, y_offset, z_offset),approach_speed,fine,Alex_Pen_ABB\WObj:=WorkSurface;
        ENDFOR

        ! Raise pen
        MoveL Offs(next_target, x_offset, y_offset, penup_offset),approach_speed,fine,Alex_Pen_ABB\WObj:=WorkSurface;

        ! Raise pen to avoid drawing of surface while moving to the new approach position
        position := pos17{1} * font_size;
        next_target.trans := position;
        MoveJ Offs(next_target, x_offset, y_offset, penup_offset),approach_speed,fine,Alex_Pen_ABB\WObj:=WorkSurface;

        ! Drop pen
        MoveL Offs(next_target, x_offset, y_offset, z_offset),approach_speed,fine,Alex_Pen_ABB\WObj:=WorkSurface;

        FOR index FROM 1 TO Dim(pos17, 1) DO
            position := pos17{index} * font_size;
            next_target.trans := position;

            MoveL Offs(next_target, x_offset, y_offset, z_offset),approach_speed,fine,Alex_Pen_ABB\WObj:=WorkSurface;
        ENDFOR

        ! Raise pen
        MoveL Offs(next_target, x_offset, y_offset, penup_offset),approach_speed,fine,Alex_Pen_ABB\WObj:=WorkSurface;

        ! Raise pen to avoid drawing of surface while moving to the new approach position
        position := pos18{1} * font_size;
        next_target.trans := position;
        MoveJ Offs(next_target, x_offset, y_offset, penup_offset),approach_speed,fine,Alex_Pen_ABB\WObj:=WorkSurface;

        ! Drop pen
        MoveL Offs(next_target, x_offset, y_offset, z_offset),approach_speed,fine,Alex_Pen_ABB\WObj:=WorkSurface;

        FOR index FROM 1 TO Dim(pos18, 1) DO
            position := pos18{index} * font_size;
            next_target.trans := position;

            MoveL Offs(next_target, x_offset, y_offset, z_offset),approach_speed,fine,Alex_Pen_ABB\WObj:=WorkSurface;
        ENDFOR

        ! Raise pen
        MoveL Offs(next_target, x_offset, y_offset, penup_offset),approach_speed,fine,Alex_Pen_ABB\WObj:=WorkSurface;

    ENDPROC

    !***********************************************************
    !
    ! Procedure VectorArt
    !   This procedure draws my vector artwork on the work surface
    !
    ! Example
    !
    !   VectorArt;
    !
    !***********************************************************
	PROC VectorArt()
	    MoveL Target_10_Appoach,v500,z10,Alex_Pen_ABB\WObj:=WorkSurface;
	    MoveL Target_10,v500,z10,Alex_Pen_ABB\WObj:=WorkSurface;
	    MoveL Target_20,v500,z10,Alex_Pen_ABB\WObj:=WorkSurface;
	    MoveL Target_30,v500,z10,Alex_Pen_ABB\WObj:=WorkSurface;
	    MoveL Target_40,v500,z10,Alex_Pen_ABB\WObj:=WorkSurface;
	    MoveL Target_50,v500,z10,Alex_Pen_ABB\WObj:=WorkSurface;
	    MoveL Target_60,v500,z10,Alex_Pen_ABB\WObj:=WorkSurface;
	    MoveL Target_70,v500,z10,Alex_Pen_ABB\WObj:=WorkSurface;
	    MoveL Target_80,v500,z10,Alex_Pen_ABB\WObj:=WorkSurface;
	    MoveL Target_90,v500,z10,Alex_Pen_ABB\WObj:=WorkSurface;
	    MoveL Target_100,v500,z10,Alex_Pen_ABB\WObj:=WorkSurface;
	    MoveL Target_110,v500,z10,Alex_Pen_ABB\WObj:=WorkSurface;
	    MoveL Target_120,v500,z10,Alex_Pen_ABB\WObj:=WorkSurface;
	    MoveL Target_130,v500,z10,Alex_Pen_ABB\WObj:=WorkSurface;
	    MoveL Target_130_Depart,v500,z10,Alex_Pen_ABB\WObj:=WorkSurface;
	ENDPROC
ENDMODULE

--- Backups/ABB_Robot/RAPID/TASK1/SYSMOD/LINKEDM.sys ---
%%%
  VERSION:1
  LANGUAGE:ENGLISH
%%%

MODULE LINKEDM (SYSMODULE)

! FOLLOWER
!     Name of electronically linked follower axis used by operator at teach pendent.
      PERS string l_f_axis_name{5}       :=  ["",  "", "", "", ""];

!     Name of the mechanical unit for follower axis.
      PERS string l_f_mecunt_n{5}  :=  ["", "", "", "", ""];

!     Linked follower axis number in the mechanical unit (first axis in mech. unit is number 1).
      PERS num l_f_axis_no{5}      :=  [0,          0,   0,  0,  0];

! MASTER
!     Name of the mechanical unit for linked master axis.
      PERS string l_m_mecunt_n{5} :=  ["", "", "", "", ""];

!     Linked master axis number in the mechanical unit (first axis in mech. unit is number 1).
!     See axis number table in documentation for different master mechanical units.
      PERS num l_m_axis_no{5}     :=  [0,  0,  0,  0,  0];

! POSITION OFFSET
!     The increase of the allowed offset position between the master and follower
!     positions, used when starting AUTO mode. As soon as the offset is decreased
!     the old configurated parameter is used.
!     Example: 3 => the configurated value of allowed offset is increased 3 times.
      PERS num offset_ratio{5}       :=  [10,  10,   10,  10,  10];

! SPEED RATIO
!     Speed_ratio used in AUTO and JOG modes [ very_slow   slow    normal    fast]
!     Value 1 = max allowed manual speed.
      CONST num speed_ratio {20}      := [0.01, 0.01, 0.01, 0.01, 0.01,
                                          0.05, 0.05, 0.05, 0.05, 0.05,
                                          0.20, 0.20, 0.20, 0.20, 0.20,
                                          1.00, 1.00, 1.00, 1.00, 1.00];

! STEP SIZE
!     Displacement position used in JOG mode for each activation of positive or
!     negative movement.                  [very_short    short   normal   long]
!     Unit degees or meter.
      CONST num displacement {20}     := [0.001, 0.001, 0.001, 0.001, 0.001,
                                          0.005, 0.005, 0.005, 0.005, 0.005,
                                          0.020, 0.020, 0.020, 0.020, 0.020,
                                          0.100, 0.100, 0.100, 0.100, 0.100];


!-------------------------------------------------------------
 PROC Linked_m ()
      Linked_m_exe ;
 ENDPROC
ENDMODULE
